Staubli VAL3: TxtFile.pjx

--- TxtFile.pjx ---
Parameters version=s7.7 stackSize=5000 millimeterUnit=true
Program file=BackupProduct.pgx
Program file=CloseFile.pgx
Program file=DeleteAlarmFile.pgx
Program file=DeleteBuffTraj.pgx
Program file=EditRecipe.pgx
Program file=GetAsyncAxis.pgx
Program file=IsAdjustTraj.pgx
Program file=IsFileOK.pgx
Program file=ReadAction.pgx
Program file=ReadCfg.pgx
Program file=ReadMatchPreset.pgx
Program file=ReadMe.pgx
Program file=ReadPartTraj.pgx
Program file=ReadPoint.pgx
Program file=ReadPreset.pgx
Program file=ReadProduct.pgx
Program file=ReadProductName.pgx
Program file=ReadSingTraj.pgx
Program file=ReadTraj.pgx
Program file=RegulaPoint.pgx
Program file=SaveAction.pgx
Program file=SaveAutoTraj.pgx
Program file=SaveCfg.pgx
Program file=SaveNewProduct.pgx
Program file=SavePartTraj.pgx
Program file=SavePreset.pgx
Program file=SaveTraj.pgx
Program file=start.pgx
Program file=stop.pgx
Data file=TxtFile.dtx
Library alias=FileDir path=Disk://FileDir/FileDir.pjx

--- TxtFile.dtx ---
public bool b7Axis
public bool b8Axis
public bool bActionWeldEnd[52]
public bool bAdjustSpEnable
public bool bAppro[6]
  [2] = true
  [3] = true
  [4] = true
  [5] = true
public bool bBypass[7]
public bool bLeave[2] = true
public bool bMatchPreset
public bool bMoreProd1Wp
public bool bMoveBack
public bool bMoveC[23]
public bool bOpenSharp
public bool bReadProduct
public bool bStartRead
public bool bSync7Axis
public bool bSync8Axis
public bool bTeachToolMode = true
public bool bTrajFilter
public bool bWeldEnable
public configRx cCfg
public frame fArray = {fatherId=fToffset[0]}
public frame fPofffset = {fatherId=fProduct[0]}
public frame fProduct = {x=-277.183, y=274.433, z=1513.292, rx=179.618, ry=-0.15, rz=0.135, fatherId=world[0]}
public frame fToffset = {fatherId=fTraj[0]}
public frame fTraj = {fatherId=fPofffset[0]}
public jointRx jAppro[6]
  [0] = {j1=37.473, j2=88.494, j3=-87.264, j4=-100.531, j5=89.054, j6=1.383}
  [1] = {j1=37.624, j2=77.945, j3=-75.448, j4=-100.7, j5=89.292, j6=2.626}
public jointRx jHome = {j1=33, j2=81, j3=-83, j4=-126, j5=90, j6=2}
public jointRx jLeave[2]
  [0] = {j1=34.791, j2=18.331, j3=101.066, j4=133.512, j5=-31.26, j6=40.017}
  [1] = {j1=38.12, j2=66.714, j3=-60.847, j4=-101.216, j5=89.968, j6=5.929}
mdesc mNomSpeed
mdesc mRun
public num nAction[51 12 2]
public num nExternalAxis[6]
num nFileBuffID
num nFileID
public num nHomeSpeed = 10
public num nMatchPreset[201 5]
public num nOpenShapeLeng
public num nPartTrajCount[100]
public num nPreset[51 5]
  [1,0] = 1
  [1,1] = 1
  [1,2] = 1
  [1,3] = 1
  [1,4] = 1
  [2,0] = 20
  [2,1] = 50
  [2,2] = 40
  [2,3] = 30
  [2,4] = 10
  [3,0] = 1
  [3,1] = 1
  [3,2] = 1
  [3,3] = 1
  [3,4] = 1
  [4,0] = 80
  [4,1] = 50
  [4,2] = 60
  [4,3] = 70
  [4,4] = 90
public num nReadCutCount
public num nReadTrajIndex = 1
public num nSingleType = 10
public num nStepLength
public num nTotalTraj = 7
public num nTrajDelay[2] = 0.3
public num nTrajIndex = 1
public num nTrajType[7]
  [0] = 10
  [1] = 10
  [2] = 10
  [3] = 10
  [4] = 10
  [5] = 10
  [6] = 9
public num nWeldActionId = 1.0863748
public pointRx pAppro[6]
  [0] = {fatherId=fArray[0]}
  [1] = {x=1202.964, y=578.195, z=257.373, rx=170.378, ry=1.129, rz=-130, fatherId=fArray[0]}
  [2] = {x=1200.953, y=-73.199, z=17.778, rx=178.998, ry=-0.002, rz=-62.905, fatherId=fArray[0]}
  [3] = {x=1200.953, y=-73.199, z=17.778, rx=178.998, ry=-0.002, rz=-62.905, fatherId=fArray[0]}
  [4] = {x=1200.953, y=-73.199, z=17.778, rx=178.998, ry=-0.002, rz=-62.905, fatherId=fArray[0]}
  [5] = {x=1200.953, y=-73.199, z=17.778, rx=178.998, ry=-0.002, rz=-62.905, fatherId=fArray[0]}
public pointRx pCut[23]
  [0] = {x=1200.196, y=-73.011, z=17.775, rx=178.998, ry=-0.002, rz=-62.905, fatherId=fArray[0]}
  [1] = {x=1199.424, y=-73.126, z=17.777, rx=178.998, ry=-0.002, rz=-62.905, fatherId=fArray[0]}
  [2] = {x=1198.755, y=-73.528, z=17.784, rx=178.998, ry=-0.002, rz=-62.905, fatherId=fArray[0]}
  [3] = {x=1198.291, y=-74.156, z=17.795, rx=178.998, ry=-0.002, rz=-62.905, fatherId=fArray[0]}
  [4] = {x=1197.953, y=-74.874, z=17.822, rx=178.998, ry=-0.002, rz=-62.905, fatherId=fArray[0]}
  [5] = {x=1197.758, y=-76.063, z=17.838, rx=178.998, ry=-0.002, rz=-62.905, fatherId=fArray[0]}
  [6] = {x=1198.207, y=-77.971, z=17.802, rx=178.998, ry=-0.002, rz=-62.905, fatherId=fArray[0]}
  [7] = {x=1199.208, y=-79.391, z=17.721, rx=178.998, ry=-0.002, rz=-62.905, fatherId=fArray[0]}
  [8] = {x=1200.754, y=-80.312, z=17.596, rx=178.998, ry=-0.002, rz=-62.905, fatherId=fArray[0]}
  [9] = {x=1202.535, y=-80.567, z=17.454, rx=178.998, ry=-0.002, rz=-62.905, fatherId=fArray[0]}
  [10] = {x=1204.293, y=-80.092, z=17.313, rx=178.998, ry=-0.002, rz=-62.905, fatherId=fArray[0]}
  [11] = {x=1205.733, y=-78.954, z=17.197, rx=178.998, ry=-0.002, rz=-62.905, fatherId=fArray[0]}
  [12] = {x=1206.543, y=-77.403, z=17.132, rx=178.998, ry=-0.002, rz=-62.905, fatherId=fArray[0]}
  [13] = {x=1206.76, y=-75.571, z=17.115, rx=178.998, ry=-0.002, rz=-62.905, fatherId=fArray[0]}
  [14] = {x=1206.253, y=-73.991, z=17.156, rx=178.998, ry=-0.002, rz=-62.905, fatherId=fArray[0]}
  [15] = {x=1205.134, y=-72.591, z=17.246, rx=178.998, ry=-0.002, rz=-62.905, fatherId=fArray[0]}
  [16] = {x=1203.479, y=-71.733, z=17.379, rx=178.998, ry=-0.002, rz=-62.905, fatherId=fArray[0]}
  [17] = {x=1201.681, y=-71.607, z=17.523, rx=178.998, ry=-0.002, rz=-62.905, fatherId=fArray[0]}
  [18] = {x=1199.977, y=-72.194, z=17.659, rx=178.998, ry=-0.002, rz=-62.905, fatherId=fArray[0]}
  [19] = {x=1198.665, y=-73.363, z=17.765, rx=178.998, ry=-0.002, rz=-62.905, fatherId=fArray[0]}
  [20] = {x=1197.953, y=-74.874, z=17.822, rx=178.998, ry=-0.002, rz=-62.905, fatherId=fArray[0]}
  [21] = {x=1197.758, y=-76.063, z=17.838, rx=178.998, ry=-0.002, rz=-62.905, fatherId=fArray[0]}
  [22] = {x=1198.207, y=-77.971, z=17.802, rx=178.998, ry=-0.002, rz=-62.905, fatherId=fArray[0]}
public pointRx pLeave[2]
  [0] = {x=1198.23, y=-78.003, z=17.8, rx=178.998, ry=-0.002, rz=-62.905, fatherId=fArray[0]}
  [1] = {fatherId=fArray[0]}
public pointRx pMoveC[23]
  [0] = {rx=-9.837, ry=-179.468, rz=-38.118, fatherId=fArray[0]}
  [1] = {fatherId=fArray[0]}
  [2] = {fatherId=fArray[0]}
  [3] = {fatherId=fArray[0]}
  [4] = {fatherId=fArray[0]}
  [5] = {fatherId=fArray[0]}
  [6] = {fatherId=fArray[0]}
  [7] = {fatherId=fArray[0]}
  [8] = {fatherId=fArray[0]}
  [9] = {fatherId=fArray[0]}
  [10] = {fatherId=fArray[0]}
  [11] = {fatherId=fArray[0]}
  [12] = {fatherId=fArray[0]}
  [13] = {fatherId=fArray[0]}
  [14] = {fatherId=fArray[0]}
  [15] = {fatherId=fArray[0]}
  [16] = {fatherId=fArray[0]}
  [17] = {fatherId=fArray[0]}
  [18] = {fatherId=fArray[0]}
  [19] = {fatherId=fArray[0]}
  [20] = {fatherId=fArray[0]}
  [21] = {fatherId=fArray[0]}
  [22] = {fatherId=fArray[0]}
public string sPresetName = "StaubliPreset"
public string sProductName = "123"
public string sTrajName[7]
  [0] = "123_1"
  [1] = "123_16"
  [2] = "123_17"
  [3] = "123_18"
  [4] = "123_19"
  [5] = "123_20"
  [6] = "123_23"
public string sTrajNameType[7]
  [0] = "123_1(不规则图形)"
  [1] = "123_16(不规则图形)"
  [2] = "123_17(不规则图形)"
  [3] = "123_18(不规则图形)"
  [4] = "123_19(不规则图形)"
  [5] = "123_20(不规则图形)"
  [6] = "123_23(同步空走路径)"
public string sTrajType[30]
  [1] = "圆-三点法(内切)"
  [2] = "圆-圆心直径(内切)"
  [3] = "三角形(内切)"
  [4] = "矩形(内切)"
  [5] = "正五边形(内切)"
  [6] = "正六边形(内切)"
  [7] = "腰形孔(内切)"
  [9] = "同步空走路径"
  [10] = "不规则图形"
  [11] = "圆-三点法(外切)"
  [12] = "圆-圆心直径(外切)"
  [13] = "三角形(外切)"
  [14] = "矩形(外切)"
  [15] = "正五边形(外切)"
  [16] = "正六边形(外切)"
  [17] = "腰形孔(外切)"
  [20] = "同步不规则图形"
  [21] = "五角星"
  [22] = "切圆管"
  [23] = "C形-圆心直径法"
  [24] = "C形-三点法"
public tool tCfg = {x=-239.363, y=-1.436, z=194.179, rx=-89.636, ry=-89.066, rz=-89.632, fatherId=flange[0]}
public tool tFileTool = {x=-239.363, y=-1.436, z=194.179, rx=-89.636, ry=-89.066, rz=-89.632, fatherId=flange[0]}
public trsf trAppro[6]
  [0] = {z=100, rx=5}
  [1] = {z=100, rx=5}
  [2] = {z=30, rx=80}
  [3] = {z=30, rx=80}
  [4] = {z=30, rx=80}
  [5] = {z=30, rx=80}
public trsf trApproAxis[6]
public trsf trArray
public trsf trAxis8Data = {y=0.001, z=1, rx=1}
public trsf trAxisData = {y=0.001, z=1, rx=1}
public trsf trBoxcar
public trsf trCorner = {x=1, z=100, rx=15, ry=5}
public trsf trCut[23]
  [0] = {z=30, rx=80}
  [1] = {x=1, z=30, rx=80}
  [2] = {x=1, z=30, rx=80}
  [3] = {z=30, rx=80}
  [4] = {x=1, z=30, rx=80}
  [5] = {x=1, z=30, rx=80}
  [6] = {x=1, z=30, rx=80}
  [7] = {x=1, z=30, rx=80}
  [8] = {x=1, z=30, rx=80}
  [9] = {x=1, z=30, rx=80}
  [10] = {x=1, z=30, rx=80}
  [11] = {x=1, z=30, rx=80}
  [12] = {x=1, z=30, rx=80}
  [13] = {x=1, z=30, rx=80}
  [14] = {x=1, z=30, rx=80}
  [15] = {x=1, z=30, rx=80}
  [16] = {x=1, z=30, rx=80}
  [17] = {x=1, z=30, rx=80}
  [18] = {x=1, z=30, rx=80}
  [19] = {x=1, z=30, rx=80}
  [20] = {x=1, z=30, rx=80}
  [21] = {x=1, z=30, rx=80}
  [22] = {x=1, z=30, rx=80}
public trsf trCutAxis[23]
public trsf trDefaultFrame
public trsf trDownLead = {ry=8}
public trsf trIODelay = {x=0.2, y=0.2}
public trsf trLeave[2]
  [0] = {z=30, rx=80}
  [1] = {z=100, rx=5}
public trsf trLeaveAxis[2]
public trsf trPointCount = {x=6, y=23, z=2}
public trsf trPresetData = {x=2000, y=200, z=32700}
public trsf trReguPara[3]
  [0] = {x=1, z=25, rx=1, ry=0.05}
  [1] = {x=1, z=25, rx=1, ry=0.05}
  [2] = {x=1, z=25, rx=1, ry=0.05}
public trsf trRegular[3]
  [0] = {x=1205.647, y=700.52, z=95.638, rx=-9.837, ry=-179.468, rz=-38.118}
  [1] = {x=1204.5, y=694.721, z=96.662, rx=-9.837, ry=-179.468, rz=-38.118}
  [2] = {x=1192.5, y=694.721, z=96.662, rx=-9.838, ry=-179.468, rz=-38.118}
public trsf trSync7Axis
public trsf trSync8Axis
public trsf trWorkplace = {x=11507, y=50, z=11507, rx=50, rz=-1}

--- start.pgx ---
program start()
  local bool l_bRes
begin
  //
  //  call ReadAction(l_bRes)
  //  call ReadPreset(l_bRes)
  //  call ReadMatchPreset("Disk://Txt/Preset1.txt","StaubliPreset",l_bRes)
  //  call ReadProduct("Disk://Txt/product.txt","Test",true,l_bRes)
  //
  //  if !l_bRes
  //    popUpMsg("Error")
  //  else
  //   // popUpMsg("OK")
  //  endIf
  //
  //  call ReadTraj("Disk://Txt/product.txt","Test",1,1,l_bRes)
  //
  //    if !l_bRes
  //    popUpMsg("Error")
  //  else
  //    popUpMsg("OK")
  //    endIf


  //  call ReadTraj("Disk://Txt/Product1.txt","1234",1,1,l_bRes)
  call ReadCfg(l_bRes)
  if !l_bRes
    disablePower()
    popUpMsg("读取配置信息出现异常")
    logMsg("读取配置信息出现异常")
  else
    //popUpMsg("读取路径OK")
  endIf


  //  //  call ReadAction(l_bRes)
  //  call ReadCfg(l_bRes)
  //  if !l_bRes
  //    popUpMsg("读取动作信息出现异常")
  //    return
  //  else
  //    popUpMsg("ok")
  //  endIf

  //    call ReadPreset(l_bRes)
  //  if !l_bRes
  //    popUpMsg("Preset ERROR")
  //    return
  //  endIf
  //
  //call ReadProduct("Disk://Txt/Recipe.txt","1008",true,l_bRes)
  //   if !l_bRes
  //    popUpMsg("Product ERROR")
  //    return
  //  endIf
  //
  //    call ReadTraj("Disk://Txt/Recipe.txt","1008",1,2,l_bRes)
  //  if !l_bRes
  //    popUpMsg("Error")
  //  endIf
  //
  //
  ////
  ////
  //
  // wait(false)

end

--- BackupProduct.pgx ---
public program BackupProduct(string x_sSFileName (dimensions=1), num x_nIndex (dimensions=1), bool x_b2Txt (dimensions=1))
begin
  call FileDir:CloseAllFile()

  //2013.10.30
  //一个工位可以选择多个产品，主要是为了法利莱
  if bMoreProd1Wp
    if $fileExists(x_sSFileName)
      if !$copy(x_sSFileName,"Disk://Txt/Product"+toString("",x_nIndex)+".txt")
        popUpMsg("复制文件出错")
        logMsg("复制文件出错")
      endIf
    endIf
    return
  endIf


  if x_b2Txt
    if $fileExists("Disk://BackUp/"+toString("",x_nIndex)+".txt")
      if !$copy("Disk://BackUp/"+toString("",x_nIndex)+".txt","Disk://Txt/product"+toString("",x_nIndex)+".txt")
        popUpMsg("复制文件出错")
      endIf
    endIf
  else
    if $fileExists(x_sSFileName)
      if !$copy(x_sSFileName,"Disk://BackUp/"+toString("",x_nIndex)+".txt")
        popUpMsg("复制文件出错")
      endIf
    endIf

  endIf















end

--- CloseFile.pgx ---
public program CloseFile()
begin


  //关闭所有文件
  call FileDir:CloseAllFile()
end

--- DeleteAlarmFile.pgx ---
public program DeleteAlarmFile()
begin
  //删除报警文件
  if $fileExists("Usr://configs/sfty.dat")
    $delete("Usr://configs/sfty.dat")

  endIf


  if $fileExists("Usr://temp/pdrv.dat")

    $delete("Usr://temp/pdrv.dat")
  endIf












end

--- DeleteBuffTraj.pgx ---
public program DeleteBuffTraj()
  local num l_nNum
  local string l_sSFileName
begin

  //2015.04.24
  //为大数据文件报错

  for l_nNum=1 to 1000

    if $fileExists("Disk://Txt/"+toString("",l_nNum)+".txt")

      $delete("Disk://Txt/"+toString("",l_nNum)+".txt")
    else
      return
    endIf


  endFor





end

--- EditRecipe.pgx ---
public program EditRecipe(num x_nTrajIndex, bool x_bDelete, bool& x_bRes)
  local num l_nTrajIndex
  local string l_sBuff
  local string l_sFileName
begin

  //对路径进行操作
  //删除路径
  //添加路径
  //修改路径


  //参数初始化
  x_bRes=false
  l_sFileName="Disk://Txt/Recipe.txt"
  if x_nTrajIndex<1
    return
  endIf
  if x_bDelete and x_nTrajIndex>nTotalTraj
    return
  endIf

  //判断文件是否存在
  if !$fileExists(l_sFileName)
    return
  endIf
  //××××××××××××××××××××××××××××××××××××××××××××××××××××××××××××××××××××
  //开始部分
  //关闭所有文件
  call FileDir:CloseAllFile()

  //文件是否可以打开
  nFileID=$fileOpen(l_sFileName,"r")
  if nFileID<0 or nFileID>9
    return
  endIf

  //文件是否可以打开
  nFileBuffID=$fileOpen("Disk://Txt/Buff.txt","w")
  if nFileBuffID<0 or nFileBuffID>9
    return
  endIf
  l_nTrajIndex=0
  while $fileGet(nFileID,l_sBuff,1)==1
    if find(l_sBuff,"BEGIN=")>=0
      l_nTrajIndex=l_nTrajIndex+1
    endIf
    if l_nTrajIndex>=x_nTrajIndex
    else
      if find(l_sBuff,"TOTALELEMENTS=")>=0
        if x_nTrajIndex==nTotalTraj+1
          l_sBuff="TOTALELEMENTS="+toString("",x_nTrajIndex)
        else
          if x_bDelete
            l_sBuff="TOTALELEMENTS="+toString("",nTotalTraj-1)
          endIf
        endIf

      endIf
      if $fileSet(nFileBuffID,l_sBuff,1)!=1
        return
      endIf
    endIf
  endWhile
  //***********************************************************************************
  //添加中间
  //关闭所有文件
  call FileDir:CloseAllFile()

  //添加文件
  if !x_bDelete
    //文件是否可以打开
    nFileID=$fileOpen("Disk://Txt/Traj.txt","r")
    if nFileID<0 or nFileID>9
      return
    endIf

    //文件是否可以打开
    nFileBuffID=$fileOpen("Disk://Txt/Buff.txt","a")
    if nFileBuffID<0 or nFileBuffID>9
      return
    endIf

    l_sBuff=""
    $fileSet(nFileBuffID,l_sBuff,1)

    while $fileGet(nFileID,l_sBuff,1)==1

      //2015.03.20
      if find(l_sBuff,"=")>=0
        if $fileSet(nFileBuffID,l_sBuff,1)!=1
          return
        endIf
      endIf
    endWhile


    l_sBuff=""
    $fileSet(nFileBuffID,l_sBuff,1)

  endIf



  //**********************************************************************
  //添加结尾
  //关闭所有文件
  call FileDir:CloseAllFile()

  //文件是否可以打开
  nFileID=$fileOpen(l_sFileName,"r")
  if nFileID<0 or nFileID>9
    return
  endIf

  //文件是否可以打开
  nFileBuffID=$fileOpen("Disk://Txt/Buff.txt","a")
  if nFileBuffID<0 or nFileBuffID>9
    return
  endIf


  l_nTrajIndex=0
  while $fileGet(nFileID,l_sBuff,1)==1
    if find(l_sBuff,"BEGIN=")>=0

      l_nTrajIndex=l_nTrajIndex+1
    endIf
    if l_nTrajIndex<=x_nTrajIndex
    else
      if $fileSet(nFileBuffID,l_sBuff,1)!=1
        return
      endIf
    endIf
  endWhile



  //××××××××××××××××××××××××××××××××××××××××××××××××××××××××××××××××××
  //重命名
  //关闭所有文件
  call FileDir:CloseAllFile()
  $delete("Disk://Txt/Recipe.txt")
  $rename("Disk://Txt/Buff.txt","Disk://Txt/Recipe.txt")

  x_bRes=true

end

--- GetAsyncAxis.pgx ---
public program GetAsyncAxis(num x_nType (dimensions=1), string& x_sText (dimensions=1), trsf& x_trAxis (dimensions=1))
  local bool l_bBool
  local num l_nBuff
  local num l_nNum
  local string l_sSBuff
begin
  if x_nType!=20 and x_nType!=9
    return
  endIf

  //把第七，第八轴给提取出来
  while find(l_sSBuff,"/")<0 and l_nNum<len(x_sText)
    l_nNum=l_nNum+1
    l_sSBuff=right(x_sText,l_nNum)
  endWhile

  l_sSBuff=right(x_sText,l_nNum-1)+",0,0,0,0"
  x_sText=left(x_sText,len(x_sText)-l_nNum)

  call FileDir:SplitTrsf(l_sSBuff,"",x_trAxis,l_bBool)














end

--- IsAdjustTraj.pgx ---
public program IsAdjustTraj(string x_sFileName, string x_sProductName, num x_nFrom, num x_nTo, bool& x_bRes)
  local string l_sFileName
  local string l_sBuff
  local num l_nNum[3]
  local trsf l_trTrsf
  local num l_nTrajIndex
  local num l_nCount
  local string l_sCount
begin

  //读取生产文件
  //生产文件格式按照LasMAN3.6格式进行


  //参数初始化
  x_bRes=false
  l_sFileName=x_sFileName
  x_nFrom=max(1,x_nFrom)
  if x_nTo<x_nFrom
    return
  endIf
  x_nTo=min(x_nTo,nTotalTraj)

  //局部变量,路径个数
  l_nTrajIndex=0
  //判断文件是否存在
  if !$fileExists(l_sFileName)
    return
  endIf

  //关闭所有文件
  call FileDir:CloseAllFile()

  //文件是否可以打开
  nFileID=$fileOpen(l_sFileName,"r")
  if nFileID<0 or nFileID>9
    return
  endIf



  //读取每行并解析
  if $fileGet(nFileID,l_sBuff,1)!=1 or find(l_sBuff,"PRODUCT="+x_sProductName)<0
    return
  endIf

  //定位到开始循环
  while l_nTrajIndex<x_nFrom
    if $fileGet(nFileID,l_sBuff,1)==1
      if find(l_sBuff,"BEGIN=")>=0
        l_nTrajIndex=l_nTrajIndex+1
      endIf
    else
      return
    endIf
  endWhile



  while $fileGet(nFileID,l_sBuff,1)==1
    if find(l_sBuff,"BEGIN=")>=0
      l_nTrajIndex=l_nTrajIndex+1
    endIf
    //查找到有关是否过滤
    while find(l_sBuff,"BYPASS=FALSE")<0
      if $fileGet(nFileID,l_sBuff,1)==1
        if find(l_sBuff,"BEGIN=")>=0
          l_nTrajIndex=l_nTrajIndex+1
        endIf
      else
        return
      endIf
    endWhile
    //判断是否到达路径条数
    if l_nTrajIndex>x_nTo
      x_bRes=true
      bStartRead=false
      return
    endIf

    //等待读取信号
    wait(bStartRead)

    //当前在读那个路径
    nReadTrajIndex=l_nTrajIndex
    nReadCutCount=0
    //读取类型
    if $fileGet(nFileID,l_sBuff,1)==1
      toNum(right(l_sBuff,len(l_sBuff)-len("CUTTYPE=")),nSingleType,x_bRes)
      if !x_bRes
        return
      endIf
    endIf


    //Array
    if $fileGet(nFileID,l_sBuff,1)==1
      call FileDir:SplitTrsf(l_sBuff,"ARRAY=",trArray,x_bRes)
      if !x_bRes
        return
      endIf
    endIf
    //对Array进行赋值
    fArray.trsf.x=fArray.trsf.y=fArray.trsf.z=fArray.trsf.rx=fArray.trsf.ry=fArray.trsf.rz=0


    //PointCount
    if $fileGet(nFileID,l_sBuff,1)==1
      call FileDir:SplitTrsf(l_sBuff,"POINTCOUNT=",trPointCount,x_bRes)
      if !x_bRes
        return
      else

        //趋近点
        //        x_bRes=trPointCount.y<500
        //        return
        //趋近点

        resize(bAppro,1,max(trPointCount.x,1))
        resize(jAppro,1,max(trPointCount.x,1))
        resize(pAppro,1,max(trPointCount.x,1))
        resize(trAppro,1,max(trPointCount.x,1))
        resize(trApproAxis,1,max(trPointCount.x,1))

        //切割点

        resize(pCut,1,min(max(trPointCount.y,1),500))
        resize(pMoveC,1,min(max(trPointCount.y,1),500))
        resize(bMoveC,1,min(max(trPointCount.y,1),500))
        resize(trCut,1,min(max(trPointCount.y,1),500))
        resize(trCutAxis,1,min(max(trPointCount.y,1),500))

        //离开点
        resize(pLeave,1,max(trPointCount.z,1))
        resize(jLeave,1,max(trPointCount.z,1))
        resize(bLeave,1,max(trPointCount.z,1))
        resize(trLeave,1,max(trPointCount.z,1))
        resize(trLeaveAxis,1,max(trPointCount.z,1))


      endIf
    endIf



    //frame
    if $fileGet(nFileID,l_sBuff,1)==1
      call FileDir:SplitTrsf(l_sBuff,"FRAME=",fTraj.trsf,x_bRes)
      if !x_bRes
        return
      endIf
    endIf


    //OFFSET
    if $fileGet(nFileID,l_sBuff,1)==1
      call FileDir:SplitTrsf(l_sBuff,"OFFSET=",fToffset.trsf,x_bRes)
      if !x_bRes
        return
      endIf
    endIf


    //Downlead
    if $fileGet(nFileID,l_sBuff,1)==1
      call FileDir:SplitTrsf(l_sBuff,"DOWNLEAD=",trDownLead,x_bRes)
      if !x_bRes
        return
      endIf
    endIf

    //WorkPlace
    if $fileGet(nFileID,l_sBuff,1)==1
      call FileDir:SplitTrsf(l_sBuff,"WORKPLACE=",trWorkplace,x_bRes)
      if !x_bRes
        return
      endIf
    endIf

    //点信息

    //×××××××××××××××××××××××××××××××××××××××××××××××××××××××××××××××××
    //趋近点
    l_nNum[0]=0
    while $fileGet(nFileID,l_sBuff,1)==1 and find(l_sBuff,"DELAYON")<0 and (find(l_sBuff,"MOVEJ=")>=0 or find(l_sBuff,"MOVEL=")>=0)
      bAppro[l_nNum[0]]=find(l_sBuff,"MOVEL")>=0
       call GetAsyncAxis(nSingleType,l_sBuff,trApproAxis[l_nNum[0]])
      if bAppro[l_nNum[0]]
        call FileDir:SplitMoveL(l_sBuff,pAppro[l_nNum[0]].trsf,trAppro[l_nNum[0]],false,x_bRes)
        if !x_bRes
          return
        endIf
      else
        call FileDir:SplitMoveJ(l_sBuff,jAppro[l_nNum[0]],trAppro[l_nNum[0]],false,x_bRes)
        if !x_bRes
          return
        endIf

      endIf
      l_nNum[0]=l_nNum[0]+1
    endWhile


    //*****************************************************************8
    if find(l_sBuff,"DELAYON=")<0
      x_bRes=false
      return
    endIf
    toNum(right(l_sBuff,len(l_sBuff)-len("DELAYON=")),nTrajDelay[0],x_bRes)
    if !x_bRes
      return
    endIf

    //*****************************************************************
    //切割点
    l_nNum[0]=0
    l_nNum[1]=1
    while $fileGet(nFileID,l_sBuff,1)==1 and find(l_sBuff,"DELAYOFF=")<0 and (find(l_sBuff,"MOVEC=")>=0 or find(l_sBuff,"MOVEL=")>=0)

      if l_nNum[0]>=500
        l_nNum[0]=0
        $fileClose(l_nNum[2])
        l_nNum[1]=l_nNum[1]+1
      endIf
      call GetAsyncAxis(nSingleType,l_sBuff,trCutAxis[l_nNum[0]])
      if l_nNum[0]==0 and trPointCount.y>500
        l_sFileName="Disk://Txt/"+toString("",l_nNum[1])+".txt"
        l_nNum[2]=$fileOpen(l_sFileName,"w")
        if l_nNum[2]<0
          x_bRes=false
          return
        endIf
        l_nCount=sel(trPointCount.y<(l_nNum[1]*500),trPointCount.y-(l_nNum[1]-1)*500,500)
        l_sCount=toString("",l_nCount)
        $fileSet(l_nNum[2],l_sCount,1)
      endIf

      if trPointCount.y>500
        $fileSet(l_nNum[2],l_sBuff,1)
      else
        bMoveC[l_nNum[0]]=find(l_sBuff,"MOVEC")>=0
        if bMoveC[l_nNum[0]]
          call FileDir:SplitMoveC(l_sBuff,pMoveC[l_nNum[0]].trsf,pCut[l_nNum[0]].trsf,trCut[l_nNum[0]],x_bRes)
          if !x_bRes
            return
          endIf
        else
          call FileDir:SplitMoveL(l_sBuff,pCut[l_nNum[0]].trsf,trCut[l_nNum[0]],true,x_bRes)
          if !x_bRes
            return
          endIf
        endIf
      endIf


      //2015.03.10
      //可自定义工艺
      if trCut[l_nNum[0]].x==0 and nSingleType!=20 and  nSingleType!=9
        call FileDir:SplitCutPreset(l_sBuff,trCutAxis[l_nNum],x_bRes)
        if !x_bRes
          return
        endIf
      endIf
      //






      l_nNum[0]=l_nNum[0]+1
    endWhile


    //************************************
    if find(l_sBuff,"DELAYOFF=")<0
      x_bRes=false
      return
    endIf

    toNum(right(l_sBuff,len(l_sBuff)-len("DELAYOFF=")),nTrajDelay[1],x_bRes)
    if !x_bRes
      return
    endIf

    //*******************************************
    //离开点
    l_nNum[0]=0
    while $fileGet(nFileID,l_sBuff,1)==1 and find(l_sBuff,"END=")<0 and (find(l_sBuff,"MOVEJ=")>=0 or find(l_sBuff,"MOVEL=")>=0)
      call GetAsyncAxis(nSingleType,l_sBuff,trLeaveAxis[l_nNum[0]])
      bLeave[l_nNum[0]]=find(l_sBuff,"MOVEL")>=0
      if bLeave[l_nNum[0]]
        call FileDir:SplitMoveL(l_sBuff,pLeave[l_nNum[0]].trsf,trLeave[l_nNum[0]],false,x_bRes)
        if !x_bRes
          return
        endIf
      else
        call FileDir:SplitMoveJ(l_sBuff,jLeave[l_nNum[0]],trLeave[l_nNum[0]],false,x_bRes)
        if !x_bRes
          return
        endIf

      endIf
      l_nNum[0]=l_nNum[0]+1
    endWhile


    call RegulaPoint(true)
    //×××××××××××××××××××××××××××××××××××××××××××××××××××××××××××××××××××
    bStartRead=false
  endWhile

  //关闭所有文件
  call FileDir:CloseAllFile()
end

--- IsFileOK.pgx ---
public program IsFileOK(bool& x_bRes (dimensions=1))
begin


  x_bRes=false

  //删除急停文件
  call DeleteAlarmFile()


  //读取动作文件是否正确
  call ReadAction(x_bRes)
  if !x_bRes
    popUpMsg("action.txt动作文件不正确")
    logMsg("action.txt动作文件不正确")
    return
  endIf

  //读取配置文件是否正确
  call ReadCfg(x_bRes)
  if !x_bRes
    popUpMsg("configure.txt配置文件不正确")
    logMsg("configure.txt配置文件不正确")
    return
  endIf


  //读取工艺文件是否正确
  call ReadPreset(x_bRes)
  if !x_bRes
    popUpMsg("preset.txt工艺文件不正确")
    logMsg("preset.txt工艺文件不正确")
    return
  endIf


end

--- ReadAction.pgx ---
public program ReadAction(bool& x_bRes (dimensions=1))
  local num l_nNum[3]
  local string l_sBuff
  local string l_sFileName
begin

  //读取动作文本
  //动作一共是200项，每项12个动作，每个动作一共是一个值
  //


  //参数初始化
  x_bRes=false
  l_sFileName="Disk://Txt/Action.txt"

  //判断文件是否存在
  if !$fileExists(l_sFileName)
    return
  endIf

  //关闭所有文件
  call FileDir:CloseAllFile()

  //文件是否可以打开
  nFileID=$fileOpen(l_sFileName,"r")
  if nFileID<0 or nFileID>9
    return
  endIf

  //对于原有值进行初始化
  for l_nNum[0]=0 to 50
    for l_nNum[1]=0 to 11
      for l_nNum[2]=0 to 1
        nAction[l_nNum[0],l_nNum[1],l_nNum[2]]=0
      endFor
    endFor
  endFor

  l_nNum[0]=l_nNum[1]=l_nNum[2]=0


  //读取每行并解析
  while $fileGet(nFileID,l_sBuff,1)==1 and l_sBuff!="" and l_nNum[0]<51
    call FileDir:SplitActionLine(l_sBuff,nAction,l_nNum[0]+1,x_bRes)
    if !x_bRes
      return
    endIf
    l_nNum[0]=l_nNum[0]+1
  endWhile
  //关闭所有文件
  call FileDir:CloseAllFile()
  x_bRes=true

end

--- ReadCfg.pgx ---
public program ReadCfg(bool& x_bRes (dimensions=1))
  local bool l_bBool[3]
  local num l_nNum[3]
  local string l_sBuff
  local string l_sFileName
  local string l_sString
  local trsf l_trBuff
begin

  //参数初始化
  x_bRes=false
  l_sFileName="Disk://Txt/Configure.txt"

  //判断文件是否存在
  if !$fileExists(l_sFileName)
    return
  endIf

  //关闭所有文件
  call FileDir:CloseAllFile()

  //文件是否可以打开
  nFileID=$fileOpen(l_sFileName,"r")
  if nFileID<0 or nFileID>9
    return
  endIf

  //读取每行并解析
  while $fileGet(nFileID,l_sBuff,1)==1

    if find(l_sBuff,"AXIS7HOME=")==0
      call FileDir:SplitTrsf(l_sBuff,"AXIS7HOME=",trAxisData,x_bRes)
      if !x_bRes
        return
      endIf
      trAxisData.rx=max(1,trAxisData.rx)
      trAxisData.z=round(sel(trAxisData.z<=1,1,trAxisData.z))
      trAxisData.y=sel(trAxisData.y<=0,0.001,trAxisData.y)
    endIf



    if find(l_sBuff,"EXTAXIS=")==0
      call FileDir:SplitTrsf(l_sBuff,"EXTAXIS=",trAxisData,x_bRes)
      if !x_bRes
        return
      endIf
      trAxisData.rx=max(1,trAxisData.rx)
      trAxisData.z=round(sel(trAxisData.z<=1,1,trAxisData.z))
      trAxisData.y=sel(trAxisData.y<=0,0.001,trAxisData.y)
    endIf


    if find(l_sBuff,"EXT8AXIS=")==0
      call FileDir:SplitTrsf(l_sBuff,"EXT8AXIS=",trAxis8Data,x_bRes)
      if !x_bRes
        return
      endIf
      trAxis8Data.rx=max(1,trAxis8Data.rx)
      trAxis8Data.z=round(sel(trAxis8Data.z<=1,1,trAxis8Data.z))
      trAxis8Data.y=sel(trAxis8Data.y<=0,0.001,trAxis8Data.y)
    endIf


    //同步七轴
    if find(l_sBuff,"7AXISSYNC=")==0
      call FileDir:SplitTrsf(l_sBuff,"7AXISSYNC=",trSync7Axis,x_bRes)
      if !x_bRes
        return
      endIf
    endIf

    //同步八轴
    if find(l_sBuff,"8AXISSYNC=")==0
      call FileDir:SplitTrsf(l_sBuff,"8AXISSYNC=",trSync8Axis,x_bRes)
      if !x_bRes
        return
      endIf

    endIf




    //********************************
    //utf-8 文件最开始有个开始符
    //
    if find(l_sBuff,"HOME=")>=0 and find(l_sBuff,"AXIS7HOME=")<0
      l_sString=left(l_sBuff,find(l_sBuff,"=")+1)
      //      if find(l_sBuff,"HOME=")==0
      call FileDir:SplitJoint(l_sBuff,l_sString,jHome,x_bRes)
      //      else
      //         call FileDir:SplitJoint(l_sBuff," HOME=",jHome,x_bRes)
      //      endIf
      if !x_bRes
        logMsg("读取configure的home出错")
        return
      else
        l_bBool[1]=true
      endIf
    endIf

    if find(l_sBuff,"TOOL=")>=0
      l_sString=left(l_sBuff,find(l_sBuff,"=")+1)
      call FileDir:SplitTrsf(l_sBuff,l_sString,tCfg.trsf,x_bRes)
      if !x_bRes
        logMsg("读取configure的tool出错")
        return
      else
        l_bBool[0]=true
      endIf

    endIf

    if find(l_sBuff,"CORNERDATA=")==0
      call FileDir:SplitTrsf(l_sBuff,"CORNERDATA=",trCorner,x_bRes)
      if !x_bRes
        return
      endIf

    endIf

    //    if find(l_sBuff,"DOWNLEADDATA=")>=0
    //      call FileDir:SplitTrsf(l_sBuff,"DOWNLEADDATA=",trDownleadData,x_bRes)
    //      if !x_bRes
    //        return
    //      endIf
    //
    //    endIf



    if find(l_sBuff,"IODELAY=")>=0
      call FileDir:SplitTrsf(l_sBuff,"IODELAY=",trIODelay,x_bRes)
      if !x_bRes
        return
      endIf

    endIf





    if find(l_sBuff,"PRESETDATA=")>=0
      call FileDir:SplitTrsf(l_sBuff,"PRESETDATA=",trPresetData,x_bRes)
      if !x_bRes
        return
      endIf

    endIf

    if find(l_sBuff,"BOXCAR=")>=0
      call FileDir:SplitTrsf(l_sBuff,"BOXCAR=",trBoxcar,x_bRes)
      if !x_bRes
        return
      endIf
    endIf






    if find(l_sBuff,"STEPLENGTH=")>=0
      toNum(right(l_sBuff,len(l_sBuff)-len("STEPLENGTH=")),nStepLength,x_bRes)
      if !x_bRes
        return
      endIf
    endIf

    if find(l_sBuff,"HOMESPEED=")>=0
      toNum(right(l_sBuff,len(l_sBuff)-len("HOMESPEED=")),nHomeSpeed,x_bRes)
      if !x_bRes
        return
      endIf
    endIf


    //读取异步第七轴使能
    if find(l_sBuff,"7AXISENABLE=")>=0
      b7Axis=find(l_sBuff,"7AXISENABLE=TRUE")>=0

    endIf

    //读取异步第八轴使能
    if find(l_sBuff,"8AXISENABLE=")>=0
      b8Axis=find(l_sBuff,"8AXISENABLE=TRUE")>=0

    endIf


    //路径是否由外部PLC来进行控制
    if find(l_sBuff,"TRAJFILTERENABLE=")>=0
      bTrajFilter=find(l_sBuff,"TRAJFILTERENABLE=TRUE")>=0

    endIf

    //拐角速度自适应
    if find(l_sBuff,"AUTOADJSUTSPEEDENABLE=")>=0
      bAdjustSpEnable=find(l_sBuff,"AUTOADJSUTSPEEDENABLE=TRUE")>=0

    endIf


    //是否是焊接
    if find(l_sBuff,"WELDENABLE=")>=0
      bWeldEnable=find(l_sBuff,"WELDENABLE=TRUE")>=0

    endIf



    //回退
    if find(l_sBuff,"MOVEBACKENABLE=")>=0
      bMoveBack=find(l_sBuff,"MOVEBACKENABLE=TRUE")>=0

    endIf


    //不拆工具示教
    if find(l_sBuff,"TEACHTOOLCALENABLE=")>=0
      bTeachToolMode=find(l_sBuff,"TEACHTOOLCALENABLE=TRUE")>=0

    endIf
    //    if find(l_sBuff,"TEACHTOOLCAlENABLE=")>=0
    //      bTeachToolMode=find(l_sBuff,"TEACHTOOLCAlENABLE=TRUE")>=0
    //
    //    endIf

    //大文件模式
    //回退
    if find(l_sBuff,"MOREPRODUCT1WORKPLACE=")>=0
      bMoreProd1Wp=find(l_sBuff,"MOREPRODUCT1WORKPLACE=TRUE")>=0
    endIf




    //*******************************************************
    //*******************************************************

    //    if find(l_sBuff,"STEPMOVEENABLE=")>=0
    //      bStepMove=find(l_sBuff,"STEPMOVEENABLE=TRUE")>=0
    //
    //    endIf
    //
    //
    if find(l_sBuff,"BIGFILEMODE=")>=0
      bMoreProd1Wp=find(l_sBuff,"BIGFILEMODE=TRUE")>=0

    endIf
    //
    //***********************************************







  endWhile
  //关闭所有文件
  call FileDir:CloseAllFile()
  bTrajFilter=false
  x_bRes=(l_bBool[1] and l_bBool[0])



end

--- ReadMatchPreset.pgx ---
public program ReadMatchPreset(string x_sFileName (dimensions=1), string x_sPresetName (dimensions=1), bool& x_bRes (dimensions=1))
  local num l_nNum[3]
  local string l_sBuff
  local string l_sFileName
begin

  //读取动作文本
  //动作一共是200项，每项12个动作，每个动作一共是一个值
  //


  //参数初始化
  x_bRes=false
  l_sFileName=x_sFileName

  //判断文件是否存在
  if !$fileExists(l_sFileName)
    return
  endIf

  //关闭所有文件
  call FileDir:CloseAllFile()

  //文件是否可以打开
  nFileID=$fileOpen(l_sFileName,"r")
  if nFileID<0 or nFileID>9
    return
  endIf

  //对于原有值进行初始化
  for l_nNum[0]=0 to 200
    for l_nNum[1]=0 to 4
      nMatchPreset[l_nNum[0],l_nNum[1]]=0
    endFor
  endFor


  l_nNum[0]=l_nNum[1]=l_nNum[2]=0


  //读取每行并解析
  if $fileGet(nFileID,l_sBuff,1)!=1 or find(l_sBuff,"PRESET="+x_sPresetName)<0
    return
  endIf

  while $fileGet(nFileID,l_sBuff,1)==1 and l_sBuff!="" and l_nNum[0]<200
    call FileDir:SplitPresetLine(l_sBuff,nMatchPreset,l_nNum[0]+1,x_bRes)
    if !x_bRes
      return
    endIf
    l_nNum[0]=l_nNum[0]+1
  endWhile

  x_bRes=true

  //关闭所有文件
  call FileDir:CloseAllFile()






end

--- ReadMe.pgx ---
program ReadMe()
begin
  //trDownLead
  //rz 圆弧度
  //ry 圆直径

  //bWeldEnable  是否焊接


end

--- ReadPartTraj.pgx ---
public program ReadPartTraj(num x_nPartId, bool& x_bRes)
  local num l_nNum[3]
  local num l_nTrajIndex
  local string l_sBuff
  local string l_sFileName
  local trsf l_trTrsf
begin

  //读取生产文件
  //生产文件格式按照LasMAN3.6格式进行


  //参数初始化
  x_bRes=false
  //  l_sFileName=x_sFileName
  //  x_nFrom=max(1,x_nFrom)
  //  if x_nTo<x_nFrom
  //    return
  //  endIf
  //  x_nTo=min(x_nTo,nTotalTraj)
  //
  //局部变量,路径个数
  //  l_nTrajIndex=0
  //判断文件是否存在
  l_sFileName="Disk://Txt/"+toString("",x_nPartId)+".txt"

  if !$fileExists(l_sFileName)
    return
  endIf

  //关闭所有文件
  call FileDir:CloseAllFile()

  //文件是否可以打开
  nFileID=$fileOpen(l_sFileName,"r")
  if nFileID<0 or nFileID>9
    return
  endIf

  $fileGet(nFileID,l_sBuff,1)
  toNum(l_sBuff,l_nNum[0],x_bRes)
  if !x_bRes or l_nNum[0]<1
    return
  endIf

  //切割点


  nPartTrajCount[x_nPartId]=l_nNum[0]
  resize(pCut,1,l_nNum[0])
  resize(pMoveC,1,l_nNum[0])
  resize(bMoveC,1,l_nNum[0])
  resize(trCut,1,l_nNum[0])

  //
  //
  //    //切割点
  l_nNum[0]=0
  while $fileGet(nFileID,l_sBuff,1)==1 and find(l_sBuff,"DELAYOFF=")<0 and (find(l_sBuff,"MOVEL=")>=0 or find(l_sBuff,"MOVEC=")>=0)
    if nPartTrajCount[x_nPartId]<=l_nNum[0]
      x_bRes=false
      return
    endIf
    bMoveC[l_nNum[0]]=find(l_sBuff,"MOVEC=")>=0
    if bMoveC[l_nNum[0]]
      call FileDir:SplitMoveC(l_sBuff,pMoveC[l_nNum[0]].trsf,pCut[l_nNum[0]].trsf,trCut[l_nNum[0]],x_bRes)
      if !x_bRes
        return
      endIf
    else
      call FileDir:SplitMoveL(l_sBuff,pCut[l_nNum[0]].trsf,trCut[l_nNum[0]],true,x_bRes)
      if !x_bRes
        return
      endIf
    endIf

    l_nNum[0]=l_nNum[0]+1
  endWhile
  x_bRes=true
  call FileDir:CloseAllFile()
end

--- ReadPoint.pgx ---
program ReadPoint(bool& x_bRes)
  local num l_nNum
  local string l_sBuff
begin
  x_bRes=false
  //*********************************************************************************************************
  //********************************************************************************************************
  //定位到开始循环

  //读取类型
  if $fileGet(nFileID,l_sBuff,1)==1
    toNum(right(l_sBuff,len(l_sBuff)-len("CUTTYPE=")),nSingleType,x_bRes)
    if !x_bRes
      return
    endIf
  endIf


  //Array
  if $fileGet(nFileID,l_sBuff,1)==1
    call FileDir:SplitTrsf(l_sBuff,"ARRAY=",trArray,x_bRes)
    if !x_bRes
      return
    endIf
  endIf
  //对Array进行赋值
  fArray.trsf.x=fArray.trsf.y=fArray.trsf.z=fArray.trsf.rx=fArray.trsf.ry=fArray.trsf.rz=0


  //PointCount
  if $fileGet(nFileID,l_sBuff,1)==1
    call FileDir:SplitTrsf(l_sBuff,"POINTCOUNT=",trPointCount,x_bRes)
    if !x_bRes
      return
    else
      //趋近点
      resize(bAppro,1,max(trPointCount.x,1))
      resize(jAppro,1,max(trPointCount.x,1))
      resize(pAppro,1,max(trPointCount.x,1))
      resize(trAppro,1,max(trPointCount.x,1))

      //切割点
      resize(pCut,1,min(max(trPointCount.y,1),500))
      resize(pMoveC,1,min(max(trPointCount.y,1),500))
      resize(bMoveC,1,min(max(trPointCount.y,1),500))
      resize(trCut,1,min(max(trPointCount.y,1),500))

      //离开点
      resize(pLeave,1,max(trPointCount.z,1))
      resize(jLeave,1,max(trPointCount.z,1))
      resize(bLeave,1,max(trPointCount.z,1))
      resize(trLeave,1,max(trPointCount.z,1))



    endIf
  endIf


  //frame
  if $fileGet(nFileID,l_sBuff,1)==1
    call FileDir:SplitTrsf(l_sBuff,"FRAME=",fTraj.trsf,x_bRes)
    if !x_bRes
      return
    endIf
  endIf


  //OFFSET
  if $fileGet(nFileID,l_sBuff,1)==1
    call FileDir:SplitTrsf(l_sBuff,"OFFSET=",fToffset.trsf,x_bRes)
    if !x_bRes
      return
    endIf
  endIf


  //Downlead
  if $fileGet(nFileID,l_sBuff,1)==1
    call FileDir:SplitTrsf(l_sBuff,"DOWNLEAD=",trDownLead,x_bRes)
    if !x_bRes
      return
    endIf
  endIf

  //WorkPlace
  if $fileGet(nFileID,l_sBuff,1)==1
    call FileDir:SplitTrsf(l_sBuff,"WORKPLACE=",trWorkplace,x_bRes)
    if !x_bRes
      return
    endIf
  endIf

  //点信息

  //×××××××××××××××××××××××××××××××××××××××××××××××××××××××××××××××××
  //趋近点
  l_nNum=0
  while $fileGet(nFileID,l_sBuff,1)==1 and find(l_sBuff,"DELAYON")<0
    bAppro[l_nNum]=find(l_sBuff,"MOVEL")>=0
    //获取外部轴
    call GetAsyncAxis(nSingleType,l_sBuff,trApproAxis[l_nNum[0]])
    if bAppro[l_nNum]
      call FileDir:SplitMoveL(l_sBuff,pAppro[l_nNum].trsf,trAppro[l_nNum],false,x_bRes)
      if !x_bRes
        return
      endIf
    else
      call FileDir:SplitMoveJ(l_sBuff,jAppro[l_nNum],trAppro[l_nNum],false,x_bRes)
      if !x_bRes
        return
      endIf

    endIf
    l_nNum=l_nNum+1
  endWhile


  //切割点
  l_nNum=0
  while $fileGet(nFileID,l_sBuff,1)==1 and find(l_sBuff,"DELAYOFF")<0
    if l_nNum==500
      bStartRead=false
      wait(bStartRead)
      l_nNum=0
    endIf

    bMoveC[l_nNum]=find(l_sBuff,"MOVEC")>=0
    //获取外部轴
    call GetAsyncAxis(nSingleType,l_sBuff,trCutAxis[l_nNum[0]])
    //
    if bMoveC[l_nNum]
      call FileDir:SplitMoveC(l_sBuff,pMoveC[l_nNum].trsf,pCut[l_nNum].trsf,trCut[l_nNum],x_bRes)
      if !x_bRes
        return
      endIf
    else
      call FileDir:SplitMoveL(l_sBuff,pCut[l_nNum].trsf,trCut[l_nNum],true,x_bRes)
      if !x_bRes
        return
      endIf

    endIf
    //2015.03.10
    //可自定义工艺
    if trCut[l_nNum[0]].x==0 and nSingleType!=20 and  nSingleType!=9
      call FileDir:SplitCutPreset(l_sBuff,trCutAxis[l_nNum],x_bRes)
      if !x_bRes
        return
      endIf
    endIf
    l_nNum=l_nNum+1
  endWhile

  //离开点
  l_nNum=0
  while $fileGet(nFileID,l_sBuff,1)==1 and find(l_sBuff,"END=")<0
    //获取外部轴
    call GetAsyncAxis(nSingleType,l_sBuff,trLeaveAxis[l_nNum[0]])
    bLeave[l_nNum]=find(l_sBuff,"MOVEL")>=0
    if bLeave[l_nNum]
      call FileDir:SplitMoveL(l_sBuff,pLeave[l_nNum].trsf,trLeave[l_nNum],false,x_bRes)
      if !x_bRes
        return
      endIf
    else
      call FileDir:SplitMoveJ(l_sBuff,jLeave[l_nNum],trLeave[l_nNum],false,x_bRes)
      if !x_bRes
        return
      endIf

    endIf
    l_nNum=l_nNum+1
  endWhile


  call RegulaPoint(true)
  //×××××××××××××××××××××××××××××××××××××××××××××××××××××××××××××××××××


end

--- ReadPreset.pgx ---
public program ReadPreset(bool& x_bRes (dimensions=1))
  local num l_nNum[3]
  local string l_sBuff
  local string l_sFileName
begin

  //读取动作文本
  //动作一共是200项，每项12个动作，每个动作一共是一个值
  //


  //参数初始化
  x_bRes=false
  l_sFileName="Disk://Txt/Preset.txt"

  //判断文件是否存在
  if !$fileExists(l_sFileName)
    return
  endIf

  //关闭所有文件
  call FileDir:CloseAllFile()

  //文件是否可以打开
  nFileID=$fileOpen(l_sFileName,"r")
  if nFileID<0 or nFileID>9
    return
  endIf

  //对于原有值进行初始化
  for l_nNum[0]=0 to 50
    for l_nNum[1]=0 to 4
      nPreset[l_nNum[0],l_nNum[1]]=0
    endFor
  endFor


  l_nNum[0]=l_nNum[1]=l_nNum[2]=0


  //读取每行并解析
  if $fileGet(nFileID,l_sBuff,1)!=1 or find(l_sBuff,"PRESET=StaubliPreset")<0
    return
  endIf

  while $fileGet(nFileID,l_sBuff,1)==1 and l_sBuff!="" and l_nNum[0]<50
    call FileDir:SplitPresetLine(l_sBuff,nPreset,l_nNum[0]+1,x_bRes)
    if !x_bRes
      return
    endIf
    l_nNum[0]=l_nNum[0]+1
  endWhile

  x_bRes=true








end

--- ReadProduct.pgx ---
public program ReadProduct(string x_sFileName, string x_sProductName, bool x_bReadTrajName, bool& x_bRes)
  local num l_nBeginEnd[2]
  local num l_nNum[3]
  local string l_sBuff
  local string l_sFileName
  local trsf l_trTrsf
  local num l_nLineCount
begin

  //读取生产文件

  //参数初始化
  x_bRes=false
  l_sFileName=x_sFileName
  nTotalTraj=0
  //判断文件是否存在
  if !$fileExists(l_sFileName) or x_sProductName==""
    return
  endIf

  //关闭所有文件
  call FileDir:CloseAllFile()

  //文件是否可以打开
  nFileID=$fileOpen(l_sFileName,"r")
  if nFileID<0 or nFileID>9
    return
  endIf


  //读取每行并解析
  //  if $fileGet(nFileID,l_sBuff,1)!=1 or l_sBuff!=("PRODUCT="+x_sProductName)
  //    return
  //  endIf
  if $fileGet(nFileID,l_sBuff,1)!=1 or find(l_sBuff,("PRODUCT="+x_sProductName))<0
    logMsg(x_sProductName+"不正确")
    return
  endIf

  //TOOL
  if $fileGet(nFileID,l_sBuff,1)==1
    call FileDir:SplitTrsf(l_sBuff,"TOOL=",tFileTool.trsf,x_bRes)
    if !x_bRes
      logMsg("工具值不正确")
      return
    endIf

    //如果工具不正确，则报错！
    if tFileTool.trsf!=tCfg.trsf
      x_bRes=false
      return
    endIf


  endIf


  //Home
  //  if $fileGet(nFileID,l_sBuff,1)==1
  //    call FileDir:SplitJoint(l_sBuff,"HOME=",jFileHome,x_bRes)
  //    if !x_bRes
  //      return
  //    endIf
  //  endIf




  //Totalelements
  if $fileGet(nFileID,l_sBuff,1)==1
    toNum(right(l_sBuff,len(l_sBuff)-len("TOTALELEMENTS=")),nTotalTraj,x_bRes)
    //判断参数合法化
    if !x_bRes or nTotalTraj<0 or (nTotalTraj!=roundDown(nTotalTraj))
      x_bRes=false
      return
    else
      if nTotalTraj==0
        resize(sTrajName,1,1)
        resize(nTrajType,1,1)
        resize(sTrajNameType,1,1)
        resize(bBypass,1,1)
        sTrajName=""
        sTrajNameType=""
        nTrajType=10
        bBypass=false
      else
        resize(sTrajName,1,nTotalTraj)
        resize(nTrajType,1,nTotalTraj)
        resize(sTrajNameType,1,nTotalTraj)
        resize(bBypass,1,nTotalTraj)
      endIf
    endIf
  endIf

  //
  //frame
  if $fileGet(nFileID,l_sBuff,1)==1
    call FileDir:SplitTrsf(l_sBuff,"FRAME=",fProduct.trsf,x_bRes)
    if !x_bRes
      logMsg("读取产品坐标系不正确")
      return
    endIf
  endIf



  //OFFSET
  if $fileGet(nFileID,l_sBuff,1)==1
    call FileDir:SplitTrsf(l_sBuff,"OFFSET=",fPofffset.trsf,x_bRes)
    if !x_bRes
      logMsg("读取产品偏移不正确")
      return
    endIf
  endIf



  //PRESET
  if $fileGet(nFileID,l_sBuff,1)==1
    bMatchPreset=!(l_sBuff=="PRESET=StaubliPreset")
    sPresetName=right(l_sBuff,len(l_sBuff)-len("PRESET="))
    //    if !x_bRes
    //      return
    //    endIf
  endIf


  if nTotalTraj==0
    x_bRes=true
    return


  endIf

  l_nBeginEnd[0]=l_nBeginEnd[1]=0









  //读取路径名
  //×××××××××××××××××××××××××××××××××××××××××××××××××××××××××××××××××
  l_nNum[0]=0
  //强制检查路径是否完整
  // if x_bReadTrajName
  if true
    while $fileGet(nFileID,l_sBuff,1)==1 and l_nNum[0]<nTotalTraj
      if find(l_sBuff,"BEGIN=")>=0
        sTrajName[l_nNum[0]]=right(l_sBuff,len(l_sBuff)-len("BEGIN="))
        l_nBeginEnd[0]=l_nBeginEnd[0]+1
      else

        //获取文件类型
        if find(l_sBuff,"CUTTYPE=")>=0
          toNum(right(l_sBuff,len(l_sBuff)-len("CUTTYPE=")),nTrajType[l_nNum[0]],x_bRes)
          if !x_bRes
            return
          else
            sTrajNameType[l_nNum[0]]=sTrajName[l_nNum[0]]+"("+sTrajType[nTrajType[l_nNum[0]]]+")"

          endIf
        else

          //获取相应的过滤
          if find(l_sBuff,"BYPASS=TRUE")>=0
            bBypass[l_nBeginEnd[1]]=true
          endIf
          if find(l_sBuff,"BYPASS=FALSE")>=0
            bBypass[l_nBeginEnd[1]]=false
          endIf

          //得到路径最后标志符
          if find(l_sBuff,"END=")>=0
            l_nBeginEnd[1]=l_nBeginEnd[1]+1
            l_nNum[0]=l_nNum[0]+1
          endIf
        endIf

      endIf

      //2016.04.22
      //对于大文件则退出
      //对于大量的打磨，3D打印进行定制
      l_nLineCount=l_nLineCount+1
      if l_nLineCount>3000
        logMsg("文件行数超过3000行")
        call FileDir:CloseAllFile()
        x_bRes=true
        return
      endIf


    endWhile
  endIf
  //×××××××××××××××××××××××××××××××××××××××××××××××××××××××××××××××××××

  //关闭所有文件
  call FileDir:CloseAllFile()
  x_bRes=(l_nBeginEnd[0]==l_nBeginEnd[1]) and (l_nBeginEnd[0]==nTotalTraj)
end

--- ReadProductName.pgx ---
public program ReadProductName(string x_sFileName (dimensions=1), bool& x_bRes (dimensions=1))
  local num l_nNum[3]
  local string l_sBuff
  local string l_sFileName
  local trsf l_trTrsf
begin

  //读取生产文件

  //参数初始化
  x_bRes=false
  l_sFileName=x_sFileName

  //判断文件是否存在
  if !$fileExists(l_sFileName)
    return
  endIf

  //关闭所有文件
  call FileDir:CloseAllFile()

  //文件是否可以打开
  nFileID=$fileOpen(l_sFileName,"r")
  if nFileID<0 or nFileID>9
    return
  endIf


  //读取每行并解析
  if $fileGet(nFileID,l_sBuff,1)!=1 or find(l_sBuff,"PRODUCT=")<0
    logMsg("读取产品名不正确")
    return
  else
    sProductName=right(l_sBuff,len(l_sBuff)-find(l_sBuff,"=")-1)
    logMsg("读取文件名："+sProductName)
    x_bRes=true
  endIf



end

--- ReadSingTraj.pgx ---
public program ReadSingTraj(string x_sTrajName, bool& x_bRes)
  local num l_nNum[3]
  local num l_nTrajIndex
  local string l_sBuff
  local string l_sFileName
  local trsf l_trTrsf
begin

  //读取生产文件
  //生产文件格式按照LasMAN3.6格式进行


  //参数初始化
  x_bRes=false
  l_sFileName="Disk://Txt/Traj.txt"

  //判断文件是否存在
  if !$fileExists(l_sFileName)
    return
  endIf

  //关闭所有文件
  call FileDir:CloseAllFile()

  //文件是否可以打开
  nFileID=$fileOpen(l_sFileName,"r")
  if nFileID<0 or nFileID>9
    return
  endIf



  //读取每行并解析
  if $fileGet(nFileID,l_sBuff,1)!=1 or find(l_sBuff,"BEGIN="+x_sTrajName)<0
    return
  endIf

  if $fileGet(nFileID,l_sBuff,1)!=1 or find(l_sBuff,"BYPASS=")<0
    return
  endIf

  call ReadPoint(x_bRes)
  //关闭所有文件
  call FileDir:CloseAllFile()
end

--- ReadTraj.pgx ---
public program ReadTraj(string x_sFileName, string x_sProductName, num x_nFrom, num x_nTo, bool& x_bRes)
  local string l_sFileName
  local string l_sBuff
  local num l_nNum[3]
  local trsf l_trTrsf
  local num l_nTrajIndex
begin

  //读取生产文件
  //生产文件格式按照LasMAN3.6格式进行


  //参数初始化
  x_bRes=false
  nReadTrajIndex=0
  l_sFileName=x_sFileName
  x_nFrom=max(1,x_nFrom)
  if x_nTo<x_nFrom
    return
  endIf
  x_nTo=min(x_nTo,nTotalTraj)


  for l_nNum=0 to size(nPartTrajCount)-1
    nPartTrajCount[l_nNum]=0
  endFor


  //判断文件是否存在
  if !$fileExists(l_sFileName)
    return
  endIf

  //关闭所有文件
  call FileDir:CloseAllFile()

  //文件是否可以打开
  nFileID=$fileOpen(l_sFileName,"r")
  if nFileID<0 or nFileID>9
    return
  endIf



  //读取每行并解析
  if $fileGet(nFileID,l_sBuff,1)!=1 or find(l_sBuff,"PRODUCT="+x_sProductName)<0
    return
  endIf




  //局部变量,路径个数
  l_nTrajIndex=0


  //定位到开始循环
  while l_nTrajIndex<x_nFrom
    if $fileGet(nFileID,l_sBuff,1)==1
      if find(l_sBuff,"BEGIN=")>=0
        l_nTrajIndex=l_nTrajIndex+1
      endIf
    else
      return
    endIf
  endWhile



  while $fileGet(nFileID,l_sBuff,1)==1
    if find(l_sBuff,"BEGIN=")>=0
      l_nTrajIndex=l_nTrajIndex+1
    endIf
    //查找到有关是否过滤
    //  while find(l_sBuff,"BYPASS=FALSE")<0 or bBypass[l_nTrajIndex-1]
    while find(l_sBuff,"BYPASS=FALSE")<0
      if find(l_sBuff,"BYPASS=TRUE")>=0
        logMsg(sProductName+"第"+toString("",l_nTrajIndex)+"条路径被过滤")
      endIf
      if $fileGet(nFileID,l_sBuff,1)==1
        if find(l_sBuff,"BEGIN=")>=0
          l_nTrajIndex=l_nTrajIndex+1
        endIf
      else
        bStartRead=false
        return
      endIf
    endWhile
    //判断是否到达路径条数
    if l_nTrajIndex>x_nTo
      x_bRes=true
      bStartRead=false
      return
    endIf

    //等待读取信号
    wait(bStartRead)

    //当前在读那个路径
    nReadTrajIndex=l_nTrajIndex
    nReadCutCount=0
    //读取类型
    if $fileGet(nFileID,l_sBuff,1)==1
      toNum(right(l_sBuff,len(l_sBuff)-len("CUTTYPE=")),nSingleType,x_bRes)
      if !x_bRes
        return
      endIf
    endIf


    //Array
    if $fileGet(nFileID,l_sBuff,1)==1
      call FileDir:SplitTrsf(l_sBuff,"ARRAY=",trArray,x_bRes)
      if !x_bRes
        return
      endIf
    endIf
    //对Array进行赋值
    fArray.trsf.x=fArray.trsf.y=fArray.trsf.z=fArray.trsf.rx=fArray.trsf.ry=fArray.trsf.rz=0


    //PointCount
    if $fileGet(nFileID,l_sBuff,1)==1
      call FileDir:SplitTrsf(l_sBuff,"POINTCOUNT=",trPointCount,x_bRes)
      if !x_bRes
        return
      endIf
      resize(bAppro,1,max(trPointCount.x,1))
      resize(jAppro,1,max(trPointCount.x,1))
      delay(0)
      resize(pAppro,1,max(trPointCount.x,1))
      resize(trAppro,1,max(trPointCount.x,1))
      resize(trApproAxis,1,max(trPointCount.x,1))

      delay(0)
      //切割点
      resize(pCut,1,min(max(trPointCount.y,1),500))
      resize(pMoveC,1,min(max(trPointCount.y,1),500))
      delay(0)
      resize(bMoveC,1,min(max(trPointCount.y,1),500))
      resize(trCut,1,min(max(trPointCount.y,1),500))
      resize(trCutAxis,1,min(max(trPointCount.y,1),500))
      delay(0)
      //离开点
      resize(pLeave,1,max(trPointCount.z,1))
      resize(jLeave,1,max(trPointCount.z,1))
      delay(0)
      resize(bLeave,1,max(trPointCount.z,1))
      resize(trLeave,1,max(trPointCount.z,1))
      resize(trLeaveAxis,1,max(trPointCount.z,1))
      delay(0)


      //强制把所有的姿态设置为same
      for l_nNum=0 to size(bAppro)-1
        pAppro[l_nNum].config=cCfg
      endFor

      for l_nNum=0 to size(bMoveC)-1
        pMoveC[l_nNum].config=pCut[l_nNum].config=cCfg
      endFor


      for l_nNum=0 to size(bLeave)-1
        pLeave[l_nNum].config=cCfg
      endFor
    endIf


    //frame
    if $fileGet(nFileID,l_sBuff,1)==1
      call FileDir:SplitTrsf(l_sBuff,"FRAME=",fTraj.trsf,x_bRes)
      if !x_bRes
        return
      endIf
    endIf


    //OFFSET
    if $fileGet(nFileID,l_sBuff,1)==1
      call FileDir:SplitTrsf(l_sBuff,"OFFSET=",fToffset.trsf,x_bRes)
      if !x_bRes
        return
      endIf
    endIf


    //Downlead
    if $fileGet(nFileID,l_sBuff,1)==1
      call FileDir:SplitTrsf(l_sBuff,"DOWNLEAD=",trDownLead,x_bRes)
      if !x_bRes
        return
      endIf
    endIf

    //WorkPlace
    if $fileGet(nFileID,l_sBuff,1)==1
      call FileDir:SplitTrsf(l_sBuff,"WORKPLACE=",trWorkplace,x_bRes)
      if !x_bRes
        return
      endIf
    endIf

    //点信息

    //×××××××××××××××××××××××××××××××××××××××××××××××××××××××××××××××××
    //趋近点
    l_nNum[0]=0
    while $fileGet(nFileID,l_sBuff,1)==1 and find(l_sBuff,"DELAYON")<0 and (find(l_sBuff,"MOVEJ=")>=0 or find(l_sBuff,"MOVEL=")>=0)
      bAppro[l_nNum[0]]=find(l_sBuff,"MOVEL")>=0
      //获取外部轴
      call GetAsyncAxis(nSingleType,l_sBuff,trApproAxis[l_nNum[0]])
      //
      if bAppro[l_nNum[0]]
        call FileDir:SplitMoveL(l_sBuff,pAppro[l_nNum[0]].trsf,trAppro[l_nNum[0]],false,x_bRes)
        if !x_bRes
          return
        endIf
      else
        call FileDir:SplitMoveJ(l_sBuff,jAppro[l_nNum[0]],trAppro[l_nNum[0]],false,x_bRes)
        if !x_bRes
          return
        endIf

      endIf
      l_nNum[0]=l_nNum[0]+1
    endWhile


    //******************************************888
    if find(l_sBuff,"DELAYON=")<0
      x_bRes=false
      return
    endIf

    toNum(right(l_sBuff,len(l_sBuff)-len("DELAYON=")),nTrajDelay[0],x_bRes)
    if !x_bRes
      return
    else

    endIf
    //**************************************************

    //切割点
    l_nNum[0]=0
    nReadCutCount=0
    while $fileGet(nFileID,l_sBuff,1)==1 and find(l_sBuff,"DELAYOFF")<0 and (find(l_sBuff,"MOVEC=")>=0 or find(l_sBuff,"MOVEL=")>=0)

      //安全机制，如果点大于的话就报错
      if nReadCutCount>trPointCount.y
        x_bRes=false
        disablePower()
        popUpMsg("读取文件出错")
        return
      endIf


      //超过500个点，则等待读取
      if l_nNum[0]>=500

        logMsg("文本已经读取"+toString("",nReadCutCount)+"点")
        wait(bStartRead)
         bStartRead=false
        l_nNum[0]=0
      endIf

      //对点进行提取
      bMoveC[l_nNum[0]]=find(l_sBuff,"MOVEC")>=0
      //获取外部轴
      call GetAsyncAxis(nSingleType,l_sBuff,trCutAxis[l_nNum[0]])
      //
      if bMoveC[l_nNum[0]]
        call FileDir:SplitMoveC(l_sBuff,pMoveC[l_nNum[0]].trsf,pCut[l_nNum[0]].trsf,trCut[l_nNum[0]],x_bRes)
        if !x_bRes
          return
        endIf
      else
        call FileDir:SplitMoveL(l_sBuff,pCut[l_nNum[0]].trsf,trCut[l_nNum[0]],true,x_bRes)
        if !x_bRes
          return
        endIf
      endIf


      //2015.03.10
      //可自定义工艺
      if trCut[l_nNum[0]].x==0 and nSingleType!=20 and nSingleType!=9
        call FileDir:SplitCutPreset(l_sBuff,trCutAxis[l_nNum],x_bRes)
        if !x_bRes
          return
        endIf
      endIf
      //








      //不规则路径，大于点数比较多的则运动
      nReadCutCount=nReadCutCount+1
      //      if round((nReadCutCount%500))>=5 and trPointCount.y>=4
      //        if nSingleType!=10
      //          x_bRes=false
      //          return
      //        endIf
      //        bStartRead=false
      //      endIf

      l_nNum[0]=l_nNum[0]+1
      if l_nNum[0]>=5
        if nSingleType!=10 and nSingleType!=20
          x_bRes=false
          logMsg("规则图形点数不对")
          disablePower()
          return
        endIf
        bStartRead=false
      endIf

    endWhile


    //************************************

    //点数不一致，则报错
    if nReadCutCount!=trPointCount.y
      disablePower()
      x_bRes=false
      logMsg(sProductName+"第"+toString("",l_nTrajIndex)+"条路径切割点个数异常")
      return
    endIf




    if find(l_sBuff,"DELAYOFF=")<0
      x_bRes=false
      return
    endIf
    toNum(right(l_sBuff,len(l_sBuff)-len("DELAYOFF=")),nTrajDelay[1],x_bRes)
    if !x_bRes
      return
    endIf

    //************************************
    //离开点
    l_nNum[0]=0
    while $fileGet(nFileID,l_sBuff,1)==1 and find(l_sBuff,"END=")<0 and (find(l_sBuff,"MOVEJ=")>=0 or find(l_sBuff,"MOVEL=")>=0)

      bLeave[l_nNum[0]]=find(l_sBuff,"MOVEL")>=0
      //获取外部轴
      call GetAsyncAxis(nSingleType,l_sBuff,trLeaveAxis[l_nNum[0]])
      //
      if bLeave[l_nNum[0]]
        call FileDir:SplitMoveL(l_sBuff,pLeave[l_nNum[0]].trsf,trLeave[l_nNum[0]],false,x_bRes)
        if !x_bRes
          return
        endIf
      else
        call FileDir:SplitMoveJ(l_sBuff,jLeave[l_nNum[0]],trLeave[l_nNum[0]],false,x_bRes)
        if !x_bRes
          return
        endIf

      endIf
      l_nNum[0]=l_nNum[0]+1
    endWhile


    call RegulaPoint(true)
    //×××××××××××××××××××××××××××××××××××××××××××××××××××××××××××××××××××
    //判断是否到达路径条数
    if l_nTrajIndex>=x_nTo
      x_bRes=true
      bStartRead=false
      return
    else
      bStartRead=false
    endIf


  endWhile
  // x_bRes=true
  bStartRead=false

end

--- RegulaPoint.pgx ---
public program RegulaPoint(bool x_backUp (dimensions=1))
  local num l_nNum
begin

  //规则图形则保存在特定的trRegular
  //规则图形的相互转换


  if nSingleType!=10 and nSingleType!=20 and nSingleType!=9
    if x_backUp

      resize(trReguPara,1,size(pCut))
      resize(trRegular,1,size(pCut))
      for l_nNum=0 to size(pCut)-1
        trRegular[l_nNum]=pCut[l_nNum].trsf
        trReguPara[l_nNum]=trCut[l_nNum]
      endFor
    else

      resize(pCut,1,size(trRegular))
      resize(pMoveC,1,size(trRegular))
      resize(bMoveC,1,size(trRegular))
      resize(trCut,1,size(trRegular))

      for l_nNum=0 to size(trRegular)-1
        pCut[l_nNum].trsf=trRegular[l_nNum]
        trCut[l_nNum]=trReguPara[l_nNum]
        bMoveC[l_nNum]=false
        trPointCount.y=size(trRegular)-1
      endFor
    endIf
  endIf






end

--- SaveAction.pgx ---
public program SaveAction(bool& x_bRes (dimensions=1))
  local num l_nNum
  local num l_nX
  local string l_sFileName
  local string l_sSBuff
begin


  //参数初始化
  x_bRes=false
  l_sFileName="Disk://Txt/Action.txt"


  //关闭所有文件
  call FileDir:CloseAllFile()


  //文件是否可以打开
  nFileID=$fileOpen(l_sFileName,"w")
  if nFileID<0 or nFileID>9
    return
  endIf


  for l_nNum=1 to 50
    l_sSBuff=toString("",l_nNum)+"="
    for l_nX=0 to 11
      l_sSBuff=l_sSBuff+toString("",nAction[l_nNum,l_nX,0])+","+toString(".2",nAction[l_nNum,l_nX,1])+";"
    endFor
    if $fileSet(nFileID,l_sSBuff,1)!=1
      return
    endIf
  endFor

  call FileDir:CloseAllFile()

  x_bRes=true

end

--- SaveAutoTraj.pgx ---
public program SaveAutoTraj()
  local num l_nNum
  local string l_sFileName
  local string l_sSBuff
begin

  //示教或者调图过程中，对于其进行自动保存





  //参数初始化
  //x_bRes=false
  l_sFileName="Disk://BackUp/Traj.txt"


  //关闭所有文件
  call FileDir:CloseAllFile()


  //文件是否可以打开
  nFileID=$fileOpen(l_sFileName,"w")
  if nFileID<0 or nFileID>9
    return
  endIf

  l_sSBuff="//Auto Save"+getDate("%d, %Y %H:%M:%S")
  if $fileSet(nFileID,l_sSBuff,1)!=1
    return
  endIf



  l_sSBuff="BEGIN="+sProductName+"_"+toString("",nTrajIndex)
  if $fileSet(nFileID,l_sSBuff,1)!=1
    return
  endIf

  l_sSBuff="BYPASS=FALSE"
  if $fileSet(nFileID,l_sSBuff,1)!=1
    return
  endIf

  l_sSBuff="CUTTYPE="+toString("",nSingleType)
  if $fileSet(nFileID,l_sSBuff,1)!=1
    return
  endIf
  l_sSBuff="ARRAY="+toString("",trArray.x)+","+toString(".3",trArray.y)+","+toString("",trArray.z)+","+toString(".3",trArray.rx)
  l_sSBuff=l_sSBuff+","+toString("",trArray.ry)+","+toString(".3",trArray.rz)
  if $fileSet(nFileID,l_sSBuff,1)!=1
    return
  endIf

  l_sSBuff="POINTCOUNT="+toString("",size(pAppro))+","+toString("",size(pCut))+","+toString("",size(pLeave))
  if $fileSet(nFileID,l_sSBuff,1)!=1
    return
  endIf


  l_sSBuff="FRAME="+toString(".3",fTraj.trsf.x)+","+toString(".3",fTraj.trsf.y)+","+toString(".3",fTraj.trsf.z)
  l_sSBuff=l_sSBuff+","+toString(".3",fTraj.trsf.rx)+","+toString(".3",fTraj.trsf.ry)+","+toString(".3",fTraj.trsf.rz)
  if $fileSet(nFileID,l_sSBuff,1)!=1
    return
  endIf

  l_sSBuff="OFFSET="+toString(".3",fToffset.trsf.x)+","+toString(".3",fToffset.trsf.y)+","+toString(".3",fToffset.trsf.z)
  l_sSBuff=l_sSBuff+","+toString(".3",fToffset.trsf.rx)+","+toString(".3",fToffset.trsf.ry)+","+toString(".3",fToffset.trsf.rz)
  if $fileSet(nFileID,l_sSBuff,1)!=1
    return
  endIf

  l_sSBuff="DOWNLEAD="+toString(".3",trDownLead.x)+","+toString(".3",trDownLead.y)+","+toString(".3",trDownLead.z)
  l_sSBuff=l_sSBuff+","+toString(".3",trDownLead.rx)+","+toString(".3",trDownLead.ry)+","+toString(".3",trDownLead.rz)
  if $fileSet(nFileID,l_sSBuff,1)!=1
    return
  endIf

  l_sSBuff="WORKPLACE="+toString(".3",trWorkplace.x)+","+toString(".3",trWorkplace.y)+","+toString(".3",trWorkplace.z)
  l_sSBuff=l_sSBuff+","+toString(".3",trWorkplace.rx)+","+toString(".3",trWorkplace.ry)+","+toString(".3",trWorkplace.rz)
  if $fileSet(nFileID,l_sSBuff,1)!=1
    return
  endIf

  //趋近点
  for l_nNum=0 to size(pAppro)-1
    if bAppro[l_nNum]
      l_sSBuff="MOVEL="+toString(".3",pAppro[l_nNum].trsf.x)+","+toString(".3",pAppro[l_nNum].trsf.y)+","+toString(".3",pAppro[l_nNum].trsf.z)+","
      l_sSBuff=l_sSBuff+toString(".3",pAppro[l_nNum].trsf.rx)+","+toString(".3",pAppro[l_nNum].trsf.ry)+","+toString(".3",pAppro[l_nNum].trsf.rz)
    else
      l_sSBuff="MOVEJ="+toString(".3",jAppro[l_nNum].j1)+","+toString(".3",jAppro[l_nNum].j2)+","+toString(".3",jAppro[l_nNum].j3)+","
      l_sSBuff=l_sSBuff+toString(".3",jAppro[l_nNum].j4)+","+toString(".3",jAppro[l_nNum].j5)+","+toString(".3",jAppro[l_nNum].j6)
    endIf
    l_sSBuff=l_sSBuff+"/"+toString("",trAppro[l_nNum].z)+","+toString("",trAppro[l_nNum].rx)
    if $fileSet(nFileID,l_sSBuff,1)!=1
      return
    endIf
  endFor

  //Delayon
  l_sSBuff="DELAYON="+toString(".3",nTrajDelay[0])
  if $fileSet(nFileID,l_sSBuff,1)!=1
    return
  endIf

  //切割点
  for l_nNum=0 to size(pCut)-1
    if bMoveC[l_nNum]
      l_sSBuff="MOVEC="
    else
      l_sSBuff="MOVEL="
    endIf
    if bMoveC[l_nNum]
      l_sSBuff=l_sSBuff+toString(".3",pMoveC[l_nNum].trsf.x)+","+toString(".3",pMoveC[l_nNum].trsf.y)+","+toString(".3",pMoveC[l_nNum].trsf.z)+","
      l_sSBuff=l_sSBuff+toString(".3",pMoveC[l_nNum].trsf.rx)+","+toString(".3",pMoveC[l_nNum].trsf.ry)+","+toString(".3",pMoveC[l_nNum].trsf.rz)+"/"
    endIf

    l_sSBuff=l_sSBuff+toString(".3",pCut[l_nNum].trsf.x)+","+toString(".3",pCut[l_nNum].trsf.y)+","+toString(".3",pCut[l_nNum].trsf.z)+","
    l_sSBuff=l_sSBuff+toString(".3",pCut[l_nNum].trsf.rx)+","+toString(".3",pCut[l_nNum].trsf.ry)+","+toString(".3",pCut[l_nNum].trsf.rz)


    l_sSBuff=l_sSBuff+"/"+toString("",trCut[l_nNum].x)+","+toString("",trCut[l_nNum].y)+"/"
    l_sSBuff=l_sSBuff+toString("",trCut[l_nNum].z)+","+toString("",trCut[l_nNum].rx)+","+toString(".2",trCut[l_nNum].ry)
    if $fileSet(nFileID,l_sSBuff,1)!=1
      return
    endIf
  endFor

  l_sSBuff="DELAYOFF="+toString(".3",nTrajDelay[1])
  if $fileSet(nFileID,l_sSBuff,1)!=1
    return
  endIf

  //离开点
  for l_nNum=0 to size(pLeave)-1
    if bLeave[l_nNum]
      l_sSBuff="MOVEL="+toString(".3",pLeave[l_nNum].trsf.x)+","+toString(".3",pLeave[l_nNum].trsf.y)+","+toString(".3",pLeave[l_nNum].trsf.z)+","
      l_sSBuff=l_sSBuff+toString(".3",pLeave[l_nNum].trsf.rx)+","+toString(".3",pLeave[l_nNum].trsf.ry)+","+toString(".3",pLeave[l_nNum].trsf.rz)
    else
      l_sSBuff="MOVEJ="+toString(".3",jLeave[l_nNum].j1)+","+toString(".3",jLeave[l_nNum].j2)+","+toString(".3",jLeave[l_nNum].j3)+","
      l_sSBuff=l_sSBuff+toString(".3",jLeave[l_nNum].j4)+","+toString(".3",jLeave[l_nNum].j5)+","+toString(".3",jLeave[l_nNum].j6)
    endIf
    l_sSBuff=l_sSBuff+"/"+toString("",trLeave[l_nNum].z)+","+toString("",trLeave[l_nNum].rx)
    if $fileSet(nFileID,l_sSBuff,1)!=1
      return
    endIf
  endFor

  //结束符
  l_sSBuff="END="+sProductName+"_"+toString("",nTrajIndex)
  if $fileSet(nFileID,l_sSBuff,1)!=1
    return
  endIf

  call FileDir:CloseAllFile()

  //x_bRes=true

end

--- SaveCfg.pgx ---
public program SaveCfg(bool& x_bRes (dimensions=1))
  local num l_nNum
  local string l_sFileName
  local string l_sSBuff
begin


  //参数初始化
  x_bRes=false
  l_sFileName="Disk://Txt/Configure.txt"


  //关闭所有文件
  call FileDir:CloseAllFile()


  //文件是否可以打开
  nFileID=$fileOpen(l_sFileName,"w")
  if nFileID<0 or nFileID>9
    return
  endIf


  //安全点
  l_sSBuff="HOME="
  l_sSBuff=l_sSBuff+toString(".3",jHome.j1)+","+toString(".3",jHome.j2)+","+toString(".3",jHome.j3)+","
  l_sSBuff=l_sSBuff+toString(".3",jHome.j4)+","+toString(".3",jHome.j5)+","+toString(".3",jHome.j6)
  if $fileSet(nFileID,l_sSBuff,1)!=1
    return
  endIf

  //工具
  l_sSBuff="TOOL="
  l_sSBuff=l_sSBuff+toString(".3",tCfg.trsf.x)+","+toString(".3",tCfg.trsf.y)+","+toString(".3",tCfg.trsf.z)+","
  l_sSBuff=l_sSBuff+toString(".3",tCfg.trsf.rx)+","+toString(".3",tCfg.trsf.ry)+","+toString(".3",tCfg.trsf.rz)
  if $fileSet(nFileID,l_sSBuff,1)!=1
    return
  endIf


  //拐角速度
  l_sSBuff="CORNERDATA="
  l_sSBuff=l_sSBuff+toString(".3",trCorner.x)+","+toString(".3",trCorner.y)+","+toString(".3",trCorner.z)+","
  l_sSBuff=l_sSBuff+toString(".3",trCorner.rx)+","+toString(".3",trCorner.ry)+","+toString(".3",trCorner.rz)
  if $fileSet(nFileID,l_sSBuff,1)!=1
    return
  endIf


  //异步7外部轴
  //l_sSBuff="AXIS7HOME="
  l_sSBuff="EXTAXIS="
  l_sSBuff=l_sSBuff+toString(".3",trAxisData.x)+","+toString(".3",trAxisData.y)+","+toString(".3",trAxisData.z)+","
  l_sSBuff=l_sSBuff+toString(".3",trAxisData.rx)+","+toString(".3",trAxisData.ry)+","+toString(".3",trAxisData.rz)
  if $fileSet(nFileID,l_sSBuff,1)!=1
    return
  endIf


  //异步8外部轴
  l_sSBuff="EXT8AXIS="
  l_sSBuff=l_sSBuff+toString(".3",trAxis8Data.x)+","+toString(".3",trAxis8Data.y)+","+toString(".3",trAxis8Data.z)+","
  l_sSBuff=l_sSBuff+toString(".3",trAxis8Data.rx)+","+toString(".3",trAxis8Data.ry)+","+toString(".3",trAxis8Data.rz)
  if $fileSet(nFileID,l_sSBuff,1)!=1
    return
  endIf



  //同步七轴
  l_sSBuff="7AXISSYNC="
  l_sSBuff=l_sSBuff+toString(".3",trSync7Axis.x)+","+toString(".3",trSync7Axis.y)+","+toString(".3",trSync7Axis.z)+","
  l_sSBuff=l_sSBuff+toString(".3",trSync7Axis.rx)+","+toString(".3",trSync7Axis.ry)+","+toString(".3",trSync7Axis.rz)
  if $fileSet(nFileID,l_sSBuff,1)!=1
    return
  endIf





  //同步八轴
  l_sSBuff="8AXISSYNC="
  l_sSBuff=l_sSBuff+toString(".3",trSync8Axis.x)+","+toString(".3",trSync8Axis.y)+","+toString(".3",trSync8Axis.z)+","
  l_sSBuff=l_sSBuff+toString(".3",trSync8Axis.rx)+","+toString(".3",trSync8Axis.ry)+","+toString(".3",trSync8Axis.rz)
  if $fileSet(nFileID,l_sSBuff,1)!=1
    return
  endIf



  //工艺参数
  l_sSBuff="PRESETDATA="
  l_sSBuff=l_sSBuff+toString(".3",trPresetData.x)+","+toString(".3",trPresetData.y)+","+toString(".3",trPresetData.z)+","
  l_sSBuff=l_sSBuff+toString(".3",trPresetData.rx)+","+toString(".3",trPresetData.ry)+","+toString(".3",trPresetData.rz)
  if $fileSet(nFileID,l_sSBuff,1)!=1
    return
  endIf



  //IO延时
  l_sSBuff="IODELAY="
  l_sSBuff=l_sSBuff+toString(".3",trIODelay.x)+","+toString(".3",trIODelay.y)+","+toString(".3",trIODelay.z)+","
  l_sSBuff=l_sSBuff+toString(".3",trIODelay.rx)+","+toString(".3",trIODelay.ry)+","+toString(".3",trIODelay.rz)
  if $fileSet(nFileID,l_sSBuff,1)!=1
    return
  endIf


  //设置BOXCAR
  l_sSBuff="BOXCAR="
  l_sSBuff=l_sSBuff+toString(".3",trBoxcar.x)+","+toString(".3",trBoxcar.y)+","+toString(".3",trBoxcar.z)+","
  l_sSBuff=l_sSBuff+toString(".3",trBoxcar.rx)+","+toString(".3",trBoxcar.ry)+","+toString(".3",trBoxcar.rz)
  if $fileSet(nFileID,l_sSBuff,1)!=1
    return
  endIf


  //步进高度
  l_sSBuff="STEPLENGTH="+toString(".3",nStepLength)

  if $fileSet(nFileID,l_sSBuff,1)!=1
    return
  endIf


  //回零速度
  l_sSBuff="HOMESPEED="+toString(".3",nHomeSpeed)

  if $fileSet(nFileID,l_sSBuff,1)!=1
    return
  endIf





  //是否存在伪七轴
  if b7Axis
    l_sSBuff="7AXISENABLE=TRUE"
  else
    l_sSBuff="7AXISENABLE=FALSE"
  endIf
  if $fileSet(nFileID,l_sSBuff,1)!=1
    return
  endIf


  //是否存在伪八轴
  if b8Axis
    l_sSBuff="8AXISENABLE=TRUE"
  else
    l_sSBuff="8AXISENABLE=FALSE"
  endIf
  if $fileSet(nFileID,l_sSBuff,1)!=1
    return
  endIf




  //是否步进
  if bTrajFilter
    l_sSBuff="TRAJFILTERENABLE=TRUE"
  else
    l_sSBuff="TRAJFILTERENABLE=FALSE"
  endIf
  if $fileSet(nFileID,l_sSBuff,1)!=1
    return
  endIf


  //boxcar是否开启
  if bAdjustSpEnable
    l_sSBuff="AUTOADJSUTSPEEDENABLE=TRUE"
  else
    l_sSBuff="AUTOADJSUTSPEEDENABLE=FALSE"
  endIf
  if $fileSet(nFileID,l_sSBuff,1)!=1
    return
  endIf


  //是否是激光焊接
  if bWeldEnable
    l_sSBuff="WELDENABLE=TRUE"
  else
    l_sSBuff="WELDENABLE=FALSE"
  endIf
  if $fileSet(nFileID,l_sSBuff,1)!=1
    return
  endIf


  //是否回退
  if bMoveBack
    l_sSBuff="MOVEBACKENABLE=TRUE"
  else
    l_sSBuff="MOVEBACKENABLE=FALSE"
  endIf
  if $fileSet(nFileID,l_sSBuff,1)!=1
    return
  endIf



  //示教工具方法
  if bTeachToolMode
    l_sSBuff="TEACHTOOLCALENABLE=TRUE"
  else
    l_sSBuff="TEACHTOOLCALENABLE=FALSE"
  endIf
  if $fileSet(nFileID,l_sSBuff,1)!=1
    return
  endIf



  //单工位多产品
  if bMoreProd1Wp
    l_sSBuff="MOREPRODUCT1WORKPLACE=TRUE"
  else
    l_sSBuff="MOREPRODUCT1WORKPLACE=FALSE"
  endIf
  if $fileSet(nFileID,l_sSBuff,1)!=1
    return
  endIf

  //单工位多产品
  if bMoreProd1Wp
    l_sSBuff="BIGFILEMODE=TRUE"
  else
    l_sSBuff="BIGFILEMODE=FALSE"
  endIf
  if $fileSet(nFileID,l_sSBuff,1)!=1
    return
  endIf


  call FileDir:CloseAllFile()

  x_bRes=true

end

--- SaveNewProduct.pgx ---
public program SaveNewProduct(bool& x_bRes (dimensions=1))
  local num l_nTrajIndex
  local string l_sFileName
  local string l_sSBuff
begin

  //建立生产文件头的文件头


  //参数初始化
  x_bRes=false
  l_sFileName="Disk://Txt/Recipe.txt"

  //××××××××××××××××××××××××××××××××××××××××××××××××××××××××××××××××××××
  //开始部分
  //关闭所有文件
  call FileDir:CloseAllFile()

  //文件是否可以打开
  nFileID=$fileOpen(l_sFileName,"w")
  if nFileID<0 or nFileID>9
    return
  endIf

  //工具
  l_sSBuff="PRODUCT=TEST"
  if $fileSet(nFileID,l_sSBuff,1)!=1
    return
  endIf


  //工具
  l_sSBuff="TOOL="
  l_sSBuff=l_sSBuff+toString(".3",tCfg.trsf.x)+","+toString(".3",tCfg.trsf.y)+","+toString(".3",tCfg.trsf.z)+","
  l_sSBuff=l_sSBuff+toString(".3",tCfg.trsf.rx)+","+toString(".3",tCfg.trsf.ry)+","+toString(".3",tCfg.trsf.rz)
  if $fileSet(nFileID,l_sSBuff,1)!=1
    return
  endIf

  l_sSBuff="TOTALELEMENTS=0"
  if $fileSet(nFileID,l_sSBuff,1)!=1
    return
  endIf

  l_sSBuff="FRAME=0,0,0,0,0,0"
  if $fileSet(nFileID,l_sSBuff,1)!=1
    return
  endIf

  l_sSBuff="OFFSET=0,0,0,0,0,0"
  if $fileSet(nFileID,l_sSBuff,1)!=1
    return
  endIf

  l_sSBuff="PRESET=StaubliPreset"
  if $fileSet(nFileID,l_sSBuff,1)!=1
    return
  endIf

  l_sSBuff=""
  if $fileSet(nFileID,l_sSBuff,1)!=1
    return
  endIf

  l_sSBuff=""
  if $fileSet(nFileID,l_sSBuff,1)!=1
    return
  endIf

  //××××××××××××××××××××××××××××××××××××××××××××××××××××××××××××××××××
  //重命名
  //关闭所有文件
  call FileDir:CloseAllFile()

  x_bRes=true

end

--- SavePartTraj.pgx ---
public program SavePartTraj(num x_nNum, bool& x_bRes)
  local num l_nNum
  local string l_sFileName
  local string l_sSBuff
begin


  //参数初始化
  x_bRes=false
  l_sFileName="Disk://Txt/"+toString("",x_nNum)+".txt"


  //关闭所有文件
  call FileDir:CloseAllFile()


  //文件是否可以打开
  nFileID=$fileOpen(l_sFileName,"w")
  if nFileID<0 or nFileID>9
    return
  endIf

  //  l_sSBuff="BEGIN="+sProductName+"_"+toString("",nTrajIndex)
  //  if $fileSet(nFileID,l_sSBuff,1)!=1
  //    return
  //  endIf
  //
  //  l_sSBuff="BYPASS=FALSE"
  //  if $fileSet(nFileID,l_sSBuff,1)!=1
  //    return
  //  endIf
  //
  //  l_sSBuff="CUTTYPE="+toString("",nSingleType)
  //  if $fileSet(nFileID,l_sSBuff,1)!=1
  //    return
  //  endIf
  //  l_sSBuff="ARRAY="+toString("",trArray.x)+","+toString(".3",trArray.y)+","+toString("",trArray.z)+","+toString(".3",trArray.rx)
  //  l_sSBuff=l_sSBuff+","+toString("",trArray.ry)+","+toString(".3",trArray.rz)
  //  if $fileSet(nFileID,l_sSBuff,1)!=1
  //    return
  //  endIf
  //
  //  l_sSBuff="POINTCOUNT="+toString("",size(pAppro))+","+toString("",size(pCut))+","+toString("",size(pLeave))
  //  if $fileSet(nFileID,l_sSBuff,1)!=1
  //    return
  //  endIf
  //
  //
  //  l_sSBuff="FRAME="+toString(".3",fTraj.trsf.x)+","+toString(".3",fTraj.trsf.y)+","+toString(".3",fTraj.trsf.z)
  //  l_sSBuff=l_sSBuff+","+toString(".3",fTraj.trsf.rx)+","+toString(".3",fTraj.trsf.ry)+","+toString(".3",fTraj.trsf.rz)
  //  if $fileSet(nFileID,l_sSBuff,1)!=1
  //    return
  //  endIf
  //
  //  l_sSBuff="OFFSET="+toString(".3",fToffset.trsf.x)+","+toString(".3",fToffset.trsf.y)+","+toString(".3",fToffset.trsf.z)
  //  l_sSBuff=l_sSBuff+","+toString(".3",fToffset.trsf.rx)+","+toString(".3",fToffset.trsf.ry)+","+toString(".3",fToffset.trsf.rz)
  //  if $fileSet(nFileID,l_sSBuff,1)!=1
  //    return
  //  endIf
  //
  //  l_sSBuff="DOWNLEAD="+toString(".3",trDownLead.x)+","+toString(".3",trDownLead.y)+","+toString(".3",trDownLead.z)
  //  l_sSBuff=l_sSBuff+","+toString(".3",trDownLead.rx)+","+toString(".3",trDownLead.ry)+","+toString(".3",trDownLead.rz)
  //  if $fileSet(nFileID,l_sSBuff,1)!=1
  //    return
  //  endIf
  //
  //  l_sSBuff="WORKPLACE="+toString(".3",trWorkplace.x)+","+toString(".3",trWorkplace.y)+","+toString(".3",trWorkplace.z)
  //  l_sSBuff=l_sSBuff+","+toString(".3",trWorkplace.rx)+","+toString(".3",trWorkplace.ry)+","+toString(".3",trWorkplace.rz)
  //  if $fileSet(nFileID,l_sSBuff,1)!=1
  //    return
  //  endIf
  //
  //  //趋近点
  //  for l_nNum=0 to size(pAppro)-1
  //    if bAppro[l_nNum]
  //      l_sSBuff="MOVEL="+toString(".3",pAppro[l_nNum].trsf.x)+","+toString(".3",pAppro[l_nNum].trsf.y)+","+toString(".3",pAppro[l_nNum].trsf.z)+","
  //      l_sSBuff=l_sSBuff+toString(".3",pAppro[l_nNum].trsf.rx)+","+toString(".3",pAppro[l_nNum].trsf.ry)+","+toString(".3",pAppro[l_nNum].trsf.rz)
  //    else
  //      l_sSBuff="MOVEJ="+toString(".3",jAppro[l_nNum].j1)+","+toString(".3",jAppro[l_nNum].j2)+","+toString(".3",jAppro[l_nNum].j3)+","
  //      l_sSBuff=l_sSBuff+toString(".3",jAppro[l_nNum].j4)+","+toString(".3",jAppro[l_nNum].j5)+","+toString(".3",jAppro[l_nNum].j6)
  //    endIf
  //    l_sSBuff=l_sSBuff+"/"+toString("",trAppro[l_nNum].z)+","+toString("",trAppro[l_nNum].rx)
  //    if $fileSet(nFileID,l_sSBuff,1)!=1
  //      return
  //    endIf
  //  endFor
  //
  //  //Delayon
  //  l_sSBuff="DELAYON="+toString(".3",nTrajDelay[0])
  //  if $fileSet(nFileID,l_sSBuff,1)!=1
  //    return
  //  endIf

  //切割点
  l_sSBuff=toString("",size(pCut))
  if $fileSet(nFileID,l_sSBuff,1)!=1
    return
  endIf
  for l_nNum=0 to size(pCut)-1
    if bMoveC[l_nNum]
      l_sSBuff="MOVEC="
    else
      l_sSBuff="MOVEL="
    endIf
    if bMoveC[l_nNum]
      l_sSBuff=l_sSBuff+toString(".3",pMoveC[l_nNum].trsf.x)+","+toString(".3",pMoveC[l_nNum].trsf.y)+","+toString(".3",pMoveC[l_nNum].trsf.z)+","
      l_sSBuff=l_sSBuff+toString(".3",pMoveC[l_nNum].trsf.rx)+","+toString(".3",pMoveC[l_nNum].trsf.ry)+","+toString(".3",pMoveC[l_nNum].trsf.rz)+"/"
    endIf

    l_sSBuff=l_sSBuff+toString(".3",pCut[l_nNum].trsf.x)+","+toString(".3",pCut[l_nNum].trsf.y)+","+toString(".3",pCut[l_nNum].trsf.z)+","
    l_sSBuff=l_sSBuff+toString(".3",pCut[l_nNum].trsf.rx)+","+toString(".3",pCut[l_nNum].trsf.ry)+","+toString(".3",pCut[l_nNum].trsf.rz)


    l_sSBuff=l_sSBuff+"/"+toString("",trCut[l_nNum].x)+","+toString("",trCut[l_nNum].y)+"/"
    l_sSBuff=l_sSBuff+toString("",trCut[l_nNum].z)+","+toString("",trCut[l_nNum].rx)+","+toString(".2",trCut[l_nNum].ry)

    //2015.03.10
    if trCut[l_nNum].x==0 and nSingleType!=20 and nSingleType!=9

      l_sSBuff=l_sSBuff+","+toString("",trCutAxis[l_nNum].rx)+","+toString("",trCutAxis[l_nNum].ry)
    endIf

    //同步外部轴
    //2014.7.25
    if nSingleType==20 or  nSingleType==9
      l_sSBuff=l_sSBuff+"/"+toString(".3",trCutAxis[l_nNum].x)+","+toString(".3",trCutAxis[l_nNum].y)

    endIf


    if $fileSet(nFileID,l_sSBuff,1)!=1
      return
    endIf
  endFor


  //  l_sSBuff="DELAYOFF="+toString(".3",nTrajDelay[1])
  //  if $fileSet(nFileID,l_sSBuff,1)!=1
  //    return
  //  endIf
  //
  //  //离开点
  //  for l_nNum=0 to size(pLeave)-1
  //    if bLeave[l_nNum]
  //      l_sSBuff="MOVEL="+toString(".3",pLeave[l_nNum].trsf.x)+","+toString(".3",pLeave[l_nNum].trsf.y)+","+toString(".3",pLeave[l_nNum].trsf.z)+","
  //      l_sSBuff=l_sSBuff+toString(".3",pLeave[l_nNum].trsf.rx)+","+toString(".3",pLeave[l_nNum].trsf.ry)+","+toString(".3",pLeave[l_nNum].trsf.rz)
  //    else
  //      l_sSBuff="MOVEJ="+toString(".3",jLeave[l_nNum].j1)+","+toString(".3",jLeave[l_nNum].j2)+","+toString(".3",jLeave[l_nNum].j3)+","
  //      l_sSBuff=l_sSBuff+toString(".3",jLeave[l_nNum].j4)+","+toString(".3",jLeave[l_nNum].j5)+","+toString(".3",jLeave[l_nNum].j6)
  //    endIf
  //    l_sSBuff=l_sSBuff+"/"+toString("",trLeave[l_nNum].z)+","+toString("",trLeave[l_nNum].rx)
  //    if $fileSet(nFileID,l_sSBuff,1)!=1
  //      return
  //    endIf
  //  endFor
  //
  //  //结束符
  //  l_sSBuff="END="+sProductName+"_"+toString("",nTrajIndex)
  //  if $fileSet(nFileID,l_sSBuff,1)!=1
  //    return
  //  endIf

  call FileDir:CloseAllFile()

  x_bRes=true

end

--- SavePreset.pgx ---
public program SavePreset(bool& x_bRes (dimensions=1))
  local num l_nNum
  local num l_nY
  local string l_sFileName
  local string l_sSBuff
begin


  //参数初始化
  x_bRes=false
  l_sFileName="Disk://Txt/Preset.txt"


  //关闭所有文件
  call FileDir:CloseAllFile()


  //文件是否可以打开
  nFileID=$fileOpen(l_sFileName,"w")
  if nFileID<0 or nFileID>9
    return
  endIf

  l_sSBuff="PRESET=StaubliPreset"
  if $fileSet(nFileID,l_sSBuff,1)!=1
    return
  endIf
  for l_nNum=1 to 50
    //最小是0，最大是100
    for l_nY=0 to 4
      nPreset[l_nNum,l_nY]=min(100,max(0,nPreset[l_nNum,l_nY]))
    endFor

    //直接输出
    l_sSBuff=toString("",nPreset[l_nNum,0])+","+toString("",nPreset[l_nNum,1])+","+toString("",nPreset[l_nNum,2])+","
    l_sSBuff=l_sSBuff+toString("",nPreset[l_nNum,3])+","+toString("",nPreset[l_nNum,4])
    if $fileSet(nFileID,l_sSBuff,1)!=1
      return
    endIf
  endFor
  call FileDir:CloseAllFile()

  x_bRes=true

end

--- SaveTraj.pgx ---
public program SaveTraj(bool& x_bRes)
  local num l_nFileID
  local num l_nNum
  local string l_sFileName
  local string l_sSBuff
begin


  //参数初始化
  x_bRes=false
  l_sFileName="Disk://Txt/Traj.txt"


  //关闭所有文件
  call FileDir:CloseAllFile()


  if size(pCut)!=size(bMoveC) or size(pCut)!=size(pMoveC) or size(pCut)!=size(trCut)
    logMsg("路径信息不一致")
    return
  endIf

  //文件是否可以打开
  nFileID=$fileOpen(l_sFileName,"w")
  if nFileID<0 or nFileID>9
    logMsg("打开TrajTXT文件出错")
    return
  endIf




  l_sSBuff="BEGIN="+sProductName+"_"+toString("",nTrajIndex)
  if $fileSet(nFileID,l_sSBuff,1)!=1
    logMsg("BEGIN文件出错")
    return
  endIf

  l_sSBuff="BYPASS=FALSE"
  if $fileSet(nFileID,l_sSBuff,1)!=1
    return
  endIf

  l_sSBuff="CUTTYPE="+toString("",nSingleType)
  if $fileSet(nFileID,l_sSBuff,1)!=1
    return
  endIf
  l_sSBuff="ARRAY="+toString("",trArray.x)+","+toString(".3",trArray.y)+","+toString("",trArray.z)+","+toString(".3",trArray.rx)
  l_sSBuff=l_sSBuff+","+toString("",trArray.ry)+","+toString(".3",trArray.rz)
  if $fileSet(nFileID,l_sSBuff,1)!=1
    return
  endIf
  if trPointCount.y<500
    l_sSBuff="POINTCOUNT="+toString("",size(pAppro))+","+toString("",size(pCut))+","+toString("",size(pLeave))
  else
    l_sSBuff="POINTCOUNT="+toString("",size(pAppro))+","+toString("",trPointCount.y)+","+toString("",size(pLeave))
  endIf

  if $fileSet(nFileID,l_sSBuff,1)!=1
    return
  endIf


  l_sSBuff="FRAME="+toString(".3",fTraj.trsf.x)+","+toString(".3",fTraj.trsf.y)+","+toString(".3",fTraj.trsf.z)
  l_sSBuff=l_sSBuff+","+toString(".3",fTraj.trsf.rx)+","+toString(".3",fTraj.trsf.ry)+","+toString(".3",fTraj.trsf.rz)
  if $fileSet(nFileID,l_sSBuff,1)!=1
    return
  endIf

  l_sSBuff="OFFSET="+toString(".3",fToffset.trsf.x)+","+toString(".3",fToffset.trsf.y)+","+toString(".3",fToffset.trsf.z)
  l_sSBuff=l_sSBuff+","+toString(".3",fToffset.trsf.rx)+","+toString(".3",fToffset.trsf.ry)+","+toString(".3",fToffset.trsf.rz)
  if $fileSet(nFileID,l_sSBuff,1)!=1
    return
  endIf

  l_sSBuff="DOWNLEAD="+toString(".3",trDownLead.x)+","+toString(".3",trDownLead.y)+","+toString(".3",trDownLead.z)
  l_sSBuff=l_sSBuff+","+toString(".3",trDownLead.rx)+","+toString(".3",trDownLead.ry)+","+toString(".3",trDownLead.rz)
  if $fileSet(nFileID,l_sSBuff,1)!=1
    return
  endIf

  l_sSBuff="WORKPLACE="+toString(".3",trWorkplace.x)+","+toString(".3",trWorkplace.y)+","+toString(".3",trWorkplace.z)
  l_sSBuff=l_sSBuff+","+toString(".3",trWorkplace.rx)+","+toString(".3",trWorkplace.ry)+","+toString(".3",trWorkplace.rz)
  if $fileSet(nFileID,l_sSBuff,1)!=1
    return
  endIf

  //趋近点
  for l_nNum=0 to size(pAppro)-1
    if bAppro[l_nNum]
      l_sSBuff="MOVEL="+toString(".3",pAppro[l_nNum].trsf.x)+","+toString(".3",pAppro[l_nNum].trsf.y)+","+toString(".3",pAppro[l_nNum].trsf.z)+","
      l_sSBuff=l_sSBuff+toString(".3",pAppro[l_nNum].trsf.rx)+","+toString(".3",pAppro[l_nNum].trsf.ry)+","+toString(".3",pAppro[l_nNum].trsf.rz)
    else
      l_sSBuff="MOVEJ="+toString(".3",jAppro[l_nNum].j1)+","+toString(".3",jAppro[l_nNum].j2)+","+toString(".3",jAppro[l_nNum].j3)+","
      l_sSBuff=l_sSBuff+toString(".3",jAppro[l_nNum].j4)+","+toString(".3",jAppro[l_nNum].j5)+","+toString(".3",jAppro[l_nNum].j6)
    endIf
    l_sSBuff=l_sSBuff+"/"+toString("",trAppro[l_nNum].z)+","+toString("",trAppro[l_nNum].rx)
    //同步外部轴
    //2014.7.25
    if nSingleType==20  or nSingleType==9
      l_sSBuff=l_sSBuff+"/"+toString(".3",trApproAxis[l_nNum].x)+","+toString(".3",trApproAxis[l_nNum].y)

    endIf


    if $fileSet(nFileID,l_sSBuff,1)!=1
      return
    endIf
  endFor

  //Delayon
  l_sSBuff="DELAYON="+toString(".3",nTrajDelay[0])
  if $fileSet(nFileID,l_sSBuff,1)!=1
    return
  endIf

  //切割点

  if trPointCount.y<=500
    for l_nNum=0 to size(pCut)-1
      if bMoveC[l_nNum]
        l_sSBuff="MOVEC="
      else
        l_sSBuff="MOVEL="
      endIf


      if bMoveC[l_nNum]
        l_sSBuff=l_sSBuff+toString(".3",pMoveC[l_nNum].trsf.x)+","+toString(".3",pMoveC[l_nNum].trsf.y)+","+toString(".3",pMoveC[l_nNum].trsf.z)+","
        l_sSBuff=l_sSBuff+toString(".3",pMoveC[l_nNum].trsf.rx)+","+toString(".3",pMoveC[l_nNum].trsf.ry)+","+toString(".3",pMoveC[l_nNum].trsf.rz)+"/"
      endIf

      //pCut
      l_sSBuff=l_sSBuff+toString(".3",pCut[l_nNum].trsf.x)+","+toString(".3",pCut[l_nNum].trsf.y)+","+toString(".3",pCut[l_nNum].trsf.z)+","
      l_sSBuff=l_sSBuff+toString(".3",pCut[l_nNum].trsf.rx)+","+toString(".3",pCut[l_nNum].trsf.ry)+","+toString(".3",pCut[l_nNum].trsf.rz)


      l_sSBuff=l_sSBuff+"/"+toString("",trCut[l_nNum].x)+","+toString("",trCut[l_nNum].y)+"/"
      l_sSBuff=l_sSBuff+toString("",trCut[l_nNum].z)+","+toString("",trCut[l_nNum].rx)+","


      //2015.03.21
      if nSingleType==20 or  nSingleType==9
        l_sSBuff=l_sSBuff+toString("",trCut[l_nNum].ry)
      else
        l_sSBuff=l_sSBuff+toString(".2",trCut[l_nNum].ry)
      endIf


      //2015.03.10
      if trCut[l_nNum].x==0 and nSingleType!=20 and nSingleType!=9

        l_sSBuff=l_sSBuff+","+toString("",trCutAxis[l_nNum].rx)+","+toString("",trCutAxis[l_nNum].ry)
      endIf


      //同步外部轴
      //2014.7.25
      if nSingleType==20 or nSingleType==9
        l_sSBuff=l_sSBuff+"/"+toString(".3",trCutAxis[l_nNum].x)+","

        //2015.03.21
        if trCutAxis[l_nNum].y==0
          l_sSBuff=l_sSBuff+"0"
        else
          l_sSBuff=l_sSBuff+toString(".3",trCutAxis[l_nNum].y)
        endIf
      endIf



      if l_sSBuff!=""
        if $fileSet(nFileID,l_sSBuff,1)!=1
          return
        endIf
      endIf

    endFor

  else
    for l_nNum=1 to roundUp(trPointCount.y/500)
      if $fileExists("Disk://Txt/"+toString("",l_nNum)+".txt")
        l_nFileID=$fileOpen("Disk://Txt/"+toString("",l_nNum)+".txt","r")
        if l_nFileID<0
          return
        endIf
        $fileGet(l_nFileID,l_sSBuff,1)
        while $fileGet(l_nFileID,l_sSBuff,1)==1
          if $fileSet(nFileID,l_sSBuff,1)!=1
            return
          endIf
        endWhile
        $fileClose(l_nFileID)
      endIf
    endFor
  endIf




  l_sSBuff="DELAYOFF="+toString(".3",nTrajDelay[1])
  if $fileSet(nFileID,l_sSBuff,1)!=1
    return
  endIf

  //离开点
  for l_nNum=0 to size(pLeave)-1
    if bLeave[l_nNum]
      l_sSBuff="MOVEL="+toString(".3",pLeave[l_nNum].trsf.x)+","+toString(".3",pLeave[l_nNum].trsf.y)+","+toString(".3",pLeave[l_nNum].trsf.z)+","
      l_sSBuff=l_sSBuff+toString(".3",pLeave[l_nNum].trsf.rx)+","+toString(".3",pLeave[l_nNum].trsf.ry)+","+toString(".3",pLeave[l_nNum].trsf.rz)
    else
      l_sSBuff="MOVEJ="+toString(".3",jLeave[l_nNum].j1)+","+toString(".3",jLeave[l_nNum].j2)+","+toString(".3",jLeave[l_nNum].j3)+","
      l_sSBuff=l_sSBuff+toString(".3",jLeave[l_nNum].j4)+","+toString(".3",jLeave[l_nNum].j5)+","+toString(".3",jLeave[l_nNum].j6)
    endIf
    l_sSBuff=l_sSBuff+"/"+toString("",trLeave[l_nNum].z)+","+toString("",trLeave[l_nNum].rx)

    //同步外部轴
    //2014.7.25
    if nSingleType==20 or nSingleType==9
      l_sSBuff=l_sSBuff+"/"+toString(".3",trLeaveAxis[l_nNum].x)+","+toString(".3",trLeaveAxis[l_nNum].y)

    endIf


    if $fileSet(nFileID,l_sSBuff,1)!=1
      return
    endIf
  endFor

  //结束符
  l_sSBuff="END="+sProductName+"_"+toString("",nTrajIndex)
  if $fileSet(nFileID,l_sSBuff,1)!=1
    return
  endIf

  call FileDir:CloseAllFile()

  x_bRes=true

end
